// TIA Portal V21 export
FUNCTION_BLOCK "FB611"   // FB611, LAD
TITLE = FB611
{ S7_Optimized_Access := 'FALSE' }
AUTHOR : PRECISE
FAMILY : PRECISE
// CIP AIR PURGING
// stored: AutoNumber false, SetENOAutomatically false
   VAR_INPUT
      CycleEnable : Bool;
      CycleRunning : Bool;
      SecPulse : Bool;
      AlwaysTrue : Bool;
      ActualTemperature : Real;
      ActualPressure : Real;
      ActualRepetition : Int;
      ParaIn : "AirPurgingInputs";
   END_VAR
   VAR_OUTPUT
      Started : Bool;
      UtilityValve : Bool;   // Air Utility
      VentValve : Bool;
      ParaOut : "AirPurgingOutputs";
      StepStatus : String[60];
      TempValve : Bool;
      TempValve_close : Bool;
   END_VAR
   VAR_IN_OUT
      Over : Bool;
      OverTemp : Bool;
      PressurePostiveTol : Real;
      PressureNegativeTol : Real;
      ControlStarted : Bool;
      TempPostiveTol : Real;
      TempNegativeTol : Real;
      HotAirValve : Bool;
      PopupSel : Bool;
      Popup : Bool;
      PopupAck : Bool;
      ControlStartedTemp : Bool;
      re_5 : Bool;
      TempReached : Bool;
      re_6 : Bool;
   END_VAR
   VAR
      ValveOnDelayPV : Int;
      ValveOffDelayPV : Int;
      RE1 : Bool;
      StepDelay { S7_SetPoint := 'True'} : "FB110";
      VentTimer { S7_SetPoint := 'True'} : "FB101";
   END_VAR
   VAR_TEMP   // added for the SCL form of the ladder/FBD networks
      _w1 : Bool;
      _w2 : Bool;
      _w3 : Bool;
      _w4 : Bool;
   END_VAR
BEGIN

REGION Network 1: Air Purging Started
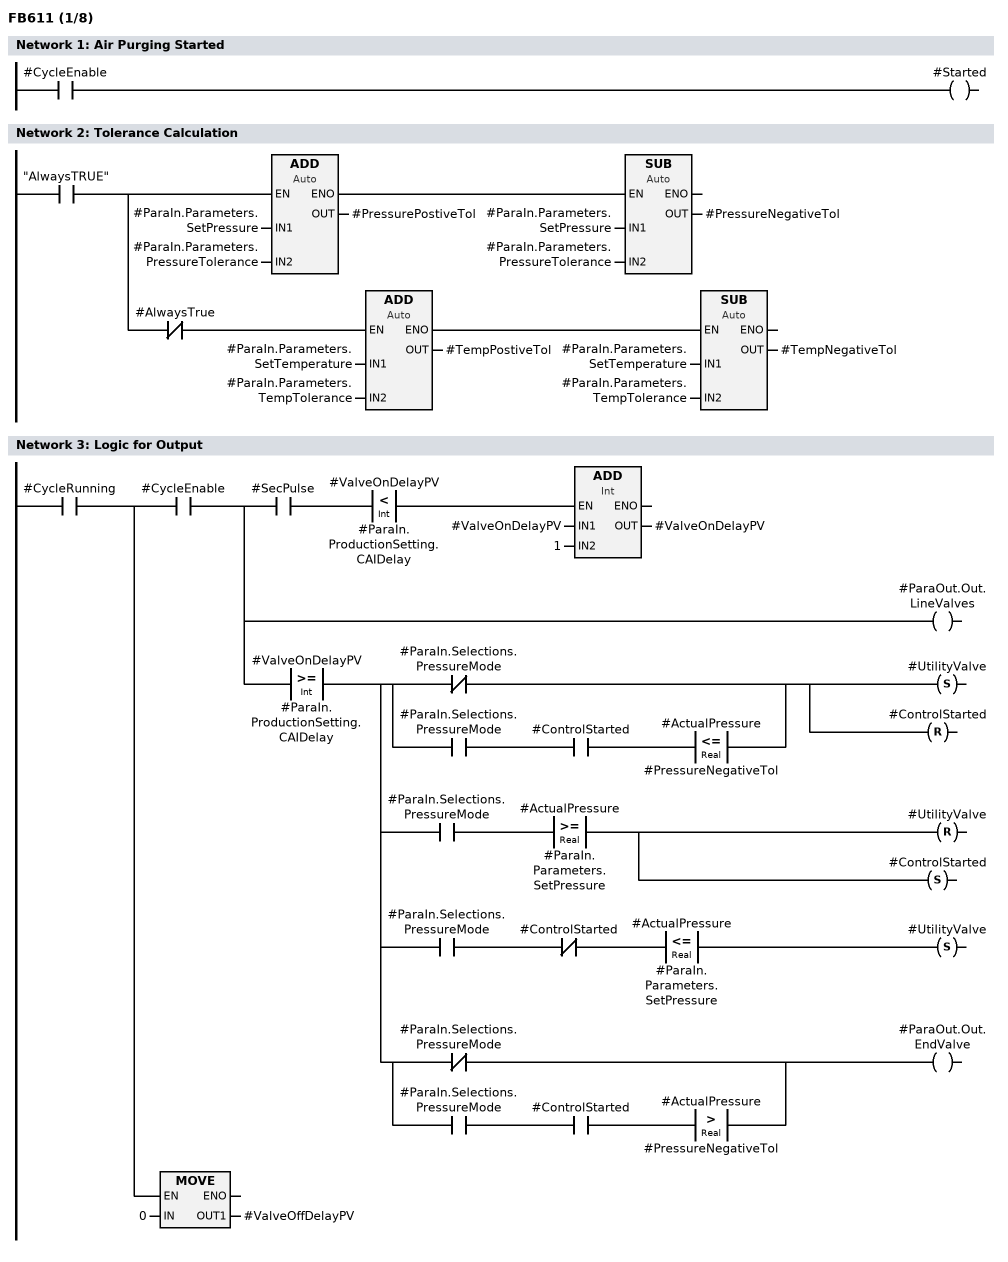
   RUNG wire#powerrail
      Contact( #CycleEnable )
      Coil( #Started )
   END_RUNG
   // the same network as SCL:
   #Started := #CycleEnable;
END_REGION

REGION Network 2: Tolerance Calculation
   RUNG wire#powerrail
      Contact( "AlwaysTRUE" )
      wire#w1
      Add(in1 := #ParaIn.Parameters.SetPressure, in2 := #ParaIn.Parameters.PressureTolerance, out => #PressurePostiveTol)
      Sub(in1 := #ParaIn.Parameters.SetPressure, in2 := #ParaIn.Parameters.PressureTolerance, out => #PressureNegativeTol)
   END_RUNG
   RUNG wire#w1
      I_Contact( #AlwaysTrue )
      Add(in1 := #ParaIn.Parameters.SetTemperature, in2 := #ParaIn.Parameters.TempTolerance, out => #TempPostiveTol)
      Sub(in1 := #ParaIn.Parameters.SetTemperature, in2 := #ParaIn.Parameters.TempTolerance, out => #TempNegativeTol)
   END_RUNG
   // the same network as SCL:
   IF "AlwaysTRUE" THEN
       #PressurePostiveTol := #ParaIn.Parameters.SetPressure + #ParaIn.Parameters.PressureTolerance;
       #PressureNegativeTol := #ParaIn.Parameters.SetPressure - #ParaIn.Parameters.PressureTolerance;
   END_IF;
   IF "AlwaysTRUE" AND NOT #AlwaysTrue THEN
       #TempPostiveTol := #ParaIn.Parameters.SetTemperature + #ParaIn.Parameters.TempTolerance;
       #TempNegativeTol := #ParaIn.Parameters.SetTemperature - #ParaIn.Parameters.TempTolerance;
   END_IF;
END_REGION

REGION Network 3: Logic for Output
   RUNG wire#powerrail
      Contact( #CycleRunning )
      wire#w1
      Contact( #CycleEnable )
      wire#w2
      Contact( #SecPulse )
      { S7_Templates := "SrcType := Int" } LT_Contact(in1 := #ValveOnDelayPV, in2 := #ParaIn.ProductionSetting.CAIDelay)
      { S7_Templates := "SrcType := Int"; S7_GenerateENO := "TRUE" } Add(in1 := #ValveOnDelayPV, in2 := 1, out => #ValveOnDelayPV)
   END_RUNG
   RUNG wire#w2
      Coil( #ParaOut.Out.LineValves )
   END_RUNG
   RUNG wire#w2
      { S7_Templates := "SrcType := Int" } GE_Contact(in1 := #ValveOnDelayPV, in2 := #ParaIn.ProductionSetting.CAIDelay)
      wire#w3
      I_Contact( #ParaIn.Selections.PressureMode )
      wire#w4
      S_Coil( #UtilityValve )
   END_RUNG
   RUNG wire#w3
      Contact( #ParaIn.Selections.PressureMode )
      Contact( #ControlStarted )
      { S7_Templates := "SrcType := Real" } LE_Contact(in1 := #ActualPressure, in2 := #PressureNegativeTol)
   END_RUNG wire#w4
   RUNG wire#w4
      R_Coil( #ControlStarted )
   END_RUNG
   RUNG wire#w3
      Contact( #ParaIn.Selections.PressureMode )
      { S7_Templates := "SrcType := Real" } GE_Contact(in1 := #ActualPressure, in2 := #ParaIn.Parameters.SetPressure)
      wire#w5
      R_Coil( #UtilityValve )
   END_RUNG
   RUNG wire#w5
      S_Coil( #ControlStarted )
   END_RUNG
   RUNG wire#w3
      Contact( #ParaIn.Selections.PressureMode )
      I_Contact( #ControlStarted )
      { S7_Templates := "SrcType := Real" } LE_Contact(in1 := #ActualPressure, in2 := #ParaIn.Parameters.SetPressure)
      S_Coil( #UtilityValve )
   END_RUNG
   RUNG wire#w3
      I_Contact( #ParaIn.Selections.PressureMode )
      wire#w6
      Coil( #ParaOut.Out.EndValve )
   END_RUNG
   RUNG wire#w3
      Contact( #ParaIn.Selections.PressureMode )
      Contact( #ControlStarted )
      { S7_Templates := "SrcType := Real" } GT_Contact(in1 := #ActualPressure, in2 := #PressureNegativeTol)
   END_RUNG wire#w6
   RUNG wire#w1
      { S7_GenerateENO := "TRUE" } Move(in := 0, out1 => #ValveOffDelayPV)
   END_RUNG
   // the same network as SCL:
   #_w1 := #CycleRunning AND #CycleEnable;
   IF #_w1 AND #SecPulse AND (#ValveOnDelayPV < #ParaIn.ProductionSetting.CAIDelay) THEN
       #ValveOnDelayPV := #ValveOnDelayPV + 1;
   END_IF;
   #ParaOut.Out.LineValves := #_w1;
   #_w2 := #_w1 AND (#ValveOnDelayPV >= #ParaIn.ProductionSetting.CAIDelay);
   IF #_w2 AND (NOT #ParaIn.Selections.PressureMode OR (#ParaIn.Selections.PressureMode AND #ControlStarted AND (#ActualPressure <= #PressureNegativeTol))) THEN
       #UtilityValve := TRUE;
       #ControlStarted := FALSE;
   END_IF;
   IF #_w2 AND #ParaIn.Selections.PressureMode AND (#ActualPressure >= #ParaIn.Parameters.SetPressure) THEN
       #UtilityValve := FALSE;
       #ControlStarted := TRUE;
   END_IF;
   IF #_w2 AND #ParaIn.Selections.PressureMode AND NOT #ControlStarted AND (#ActualPressure <= #ParaIn.Parameters.SetPressure) THEN
       #UtilityValve := TRUE;
   END_IF;
   #ParaOut.Out.EndValve := #_w2 AND (NOT #ParaIn.Selections.PressureMode OR (#ParaIn.Selections.PressureMode AND #ControlStarted AND (#ActualPressure > #PressureNegativeTol)));
   IF #CycleRunning THEN #ValveOffDelayPV := 0; END_IF;
END_REGION

REGION Network 4: Logic for Output Air Purging Sel
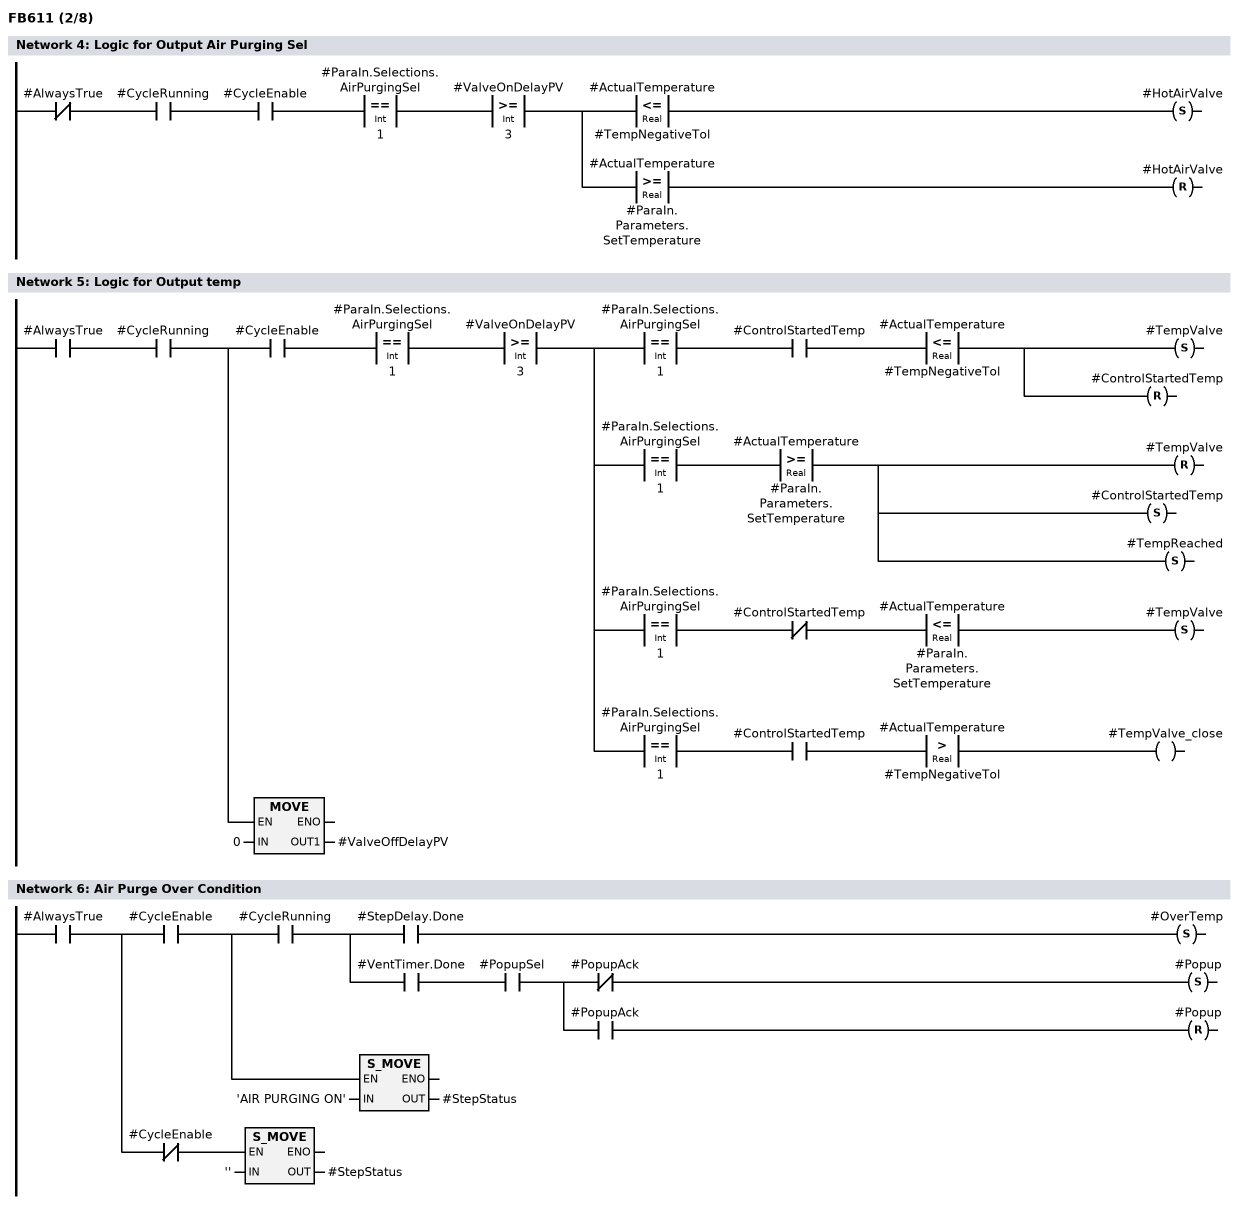
   RUNG wire#powerrail
      I_Contact( #AlwaysTrue )
      Contact( #CycleRunning )
      Contact( #CycleEnable )
      { S7_Templates := "SrcType := Int" } EQ_Contact(in1 := #ParaIn.Selections.AirPurgingSel, in2 := 1)
      { S7_Templates := "SrcType := Int" } GE_Contact(in1 := #ValveOnDelayPV, in2 := 3)
      wire#w1
      { S7_Templates := "SrcType := Real" } LE_Contact(in1 := #ActualTemperature, in2 := #TempNegativeTol)
      S_Coil( #HotAirValve )
   END_RUNG
   RUNG wire#w1
      { S7_Templates := "SrcType := Real" } GE_Contact(in1 := #ActualTemperature, in2 := #ParaIn.Parameters.SetTemperature)
      R_Coil( #HotAirValve )
   END_RUNG
   // the same network as SCL:
   #_w1 := NOT #AlwaysTrue AND #CycleRunning AND #CycleEnable AND (#ParaIn.Selections.AirPurgingSel = 1) AND (#ValveOnDelayPV >= 3);
   IF #_w1 AND (#ActualTemperature <= #TempNegativeTol) THEN #HotAirValve := TRUE; END_IF;
   IF #_w1 AND (#ActualTemperature >= #ParaIn.Parameters.SetTemperature) THEN #HotAirValve := FALSE; END_IF;
END_REGION

REGION Network 5: Logic for Output temp
   RUNG wire#powerrail
      Contact( #AlwaysTrue )
      Contact( #CycleRunning )
      wire#w1
      Contact( #CycleEnable )
      { S7_Templates := "SrcType := Int" } EQ_Contact(in1 := #ParaIn.Selections.AirPurgingSel, in2 := 1)
      { S7_Templates := "SrcType := Int" } GE_Contact(in1 := #ValveOnDelayPV, in2 := 3)
      wire#w2
      { S7_Templates := "SrcType := Int" } EQ_Contact(in1 := #ParaIn.Selections.AirPurgingSel, in2 := 1)
      Contact( #ControlStartedTemp )
      { S7_Templates := "SrcType := Real" } LE_Contact(in1 := #ActualTemperature, in2 := #TempNegativeTol)
      wire#w3
      S_Coil( #TempValve )
   END_RUNG
   RUNG wire#w3
      R_Coil( #ControlStartedTemp )
   END_RUNG
   RUNG wire#w2
      { S7_Templates := "SrcType := Int" } EQ_Contact(in1 := #ParaIn.Selections.AirPurgingSel, in2 := 1)
      { S7_Templates := "SrcType := Real" } GE_Contact(in1 := #ActualTemperature, in2 := #ParaIn.Parameters.SetTemperature)
      wire#w4
      R_Coil( #TempValve )
   END_RUNG
   RUNG wire#w4
      S_Coil( #ControlStartedTemp )
   END_RUNG
   RUNG wire#w4
      S_Coil( #TempReached )
   END_RUNG
   RUNG wire#w2
      { S7_Templates := "SrcType := Int" } EQ_Contact(in1 := #ParaIn.Selections.AirPurgingSel, in2 := 1)
      I_Contact( #ControlStartedTemp )
      { S7_Templates := "SrcType := Real" } LE_Contact(in1 := #ActualTemperature, in2 := #ParaIn.Parameters.SetTemperature)
      S_Coil( #TempValve )
   END_RUNG
   RUNG wire#w2
      { S7_Templates := "SrcType := Int" } EQ_Contact(in1 := #ParaIn.Selections.AirPurgingSel, in2 := 1)
      Contact( #ControlStartedTemp )
      { S7_Templates := "SrcType := Real" } GT_Contact(in1 := #ActualTemperature, in2 := #TempNegativeTol)
      Coil( #TempValve_close )
   END_RUNG
   RUNG wire#w1
      { S7_GenerateENO := "TRUE" } Move(in := 0, out1 => #ValveOffDelayPV)
   END_RUNG
   // the same network as SCL:
   #_w1 := #AlwaysTrue AND #CycleRunning;
   #_w2 := #_w1 AND #CycleEnable AND (#ParaIn.Selections.AirPurgingSel = 1) AND (#ValveOnDelayPV >= 3);
   IF #_w2 AND (#ParaIn.Selections.AirPurgingSel = 1) AND #ControlStartedTemp AND (#ActualTemperature <= #TempNegativeTol) THEN
       #TempValve := TRUE;
       #ControlStartedTemp := FALSE;
   END_IF;
   IF #_w2 AND (#ParaIn.Selections.AirPurgingSel = 1) AND (#ActualTemperature >= #ParaIn.Parameters.SetTemperature) THEN
       #TempValve := FALSE;
       #ControlStartedTemp := TRUE;
       #TempReached := TRUE;
   END_IF;
   IF #_w2 AND (#ParaIn.Selections.AirPurgingSel = 1) AND NOT #ControlStartedTemp AND (#ActualTemperature <= #ParaIn.Parameters.SetTemperature) THEN
       #TempValve := TRUE;
   END_IF;
   #TempValve_close := #_w2 AND (#ParaIn.Selections.AirPurgingSel = 1) AND #ControlStartedTemp AND (#ActualTemperature > #TempNegativeTol);
   IF #_w1 THEN #ValveOffDelayPV := 0; END_IF;
END_REGION

REGION Network 6: Air Purge Over Condition
   RUNG wire#powerrail
      Contact( #AlwaysTrue )
      wire#w1
      Contact( #CycleEnable )
      wire#w2
      Contact( #CycleRunning )
      wire#w3
      Contact( #StepDelay.Done )
      S_Coil( #OverTemp )
   END_RUNG
   RUNG wire#w3
      Contact( #VentTimer.Done )
      Contact( #PopupSel )
      wire#w4
      I_Contact( #PopupAck )
      S_Coil( #Popup )
   END_RUNG
   RUNG wire#w4
      Contact( #PopupAck )
      R_Coil( #Popup )
   END_RUNG
   RUNG wire#w2
      S_Move(in := 'AIR PURGING ON', out => #StepStatus)
   END_RUNG
   RUNG wire#w1
      I_Contact( #CycleEnable )
      S_Move(in := '', out => #StepStatus)
   END_RUNG
   // the same network as SCL:
   #_w1 := #AlwaysTrue AND #CycleEnable;
   #_w2 := #_w1 AND #CycleRunning;
   IF #_w2 AND #StepDelay.Done THEN #OverTemp := TRUE; END_IF;
   #_w3 := #_w2 AND #VentTimer.Done AND #PopupSel;
   IF #_w3 AND NOT #PopupAck THEN #Popup := TRUE; END_IF;
   IF #_w3 AND #PopupAck THEN #Popup := FALSE; END_IF;
   IF #_w1 THEN #StepStatus := 'AIR PURGING ON'; END_IF;
   IF #AlwaysTrue AND NOT #CycleEnable THEN #StepStatus := ''; END_IF;
END_REGION

REGION Network 7: Air Purge Over
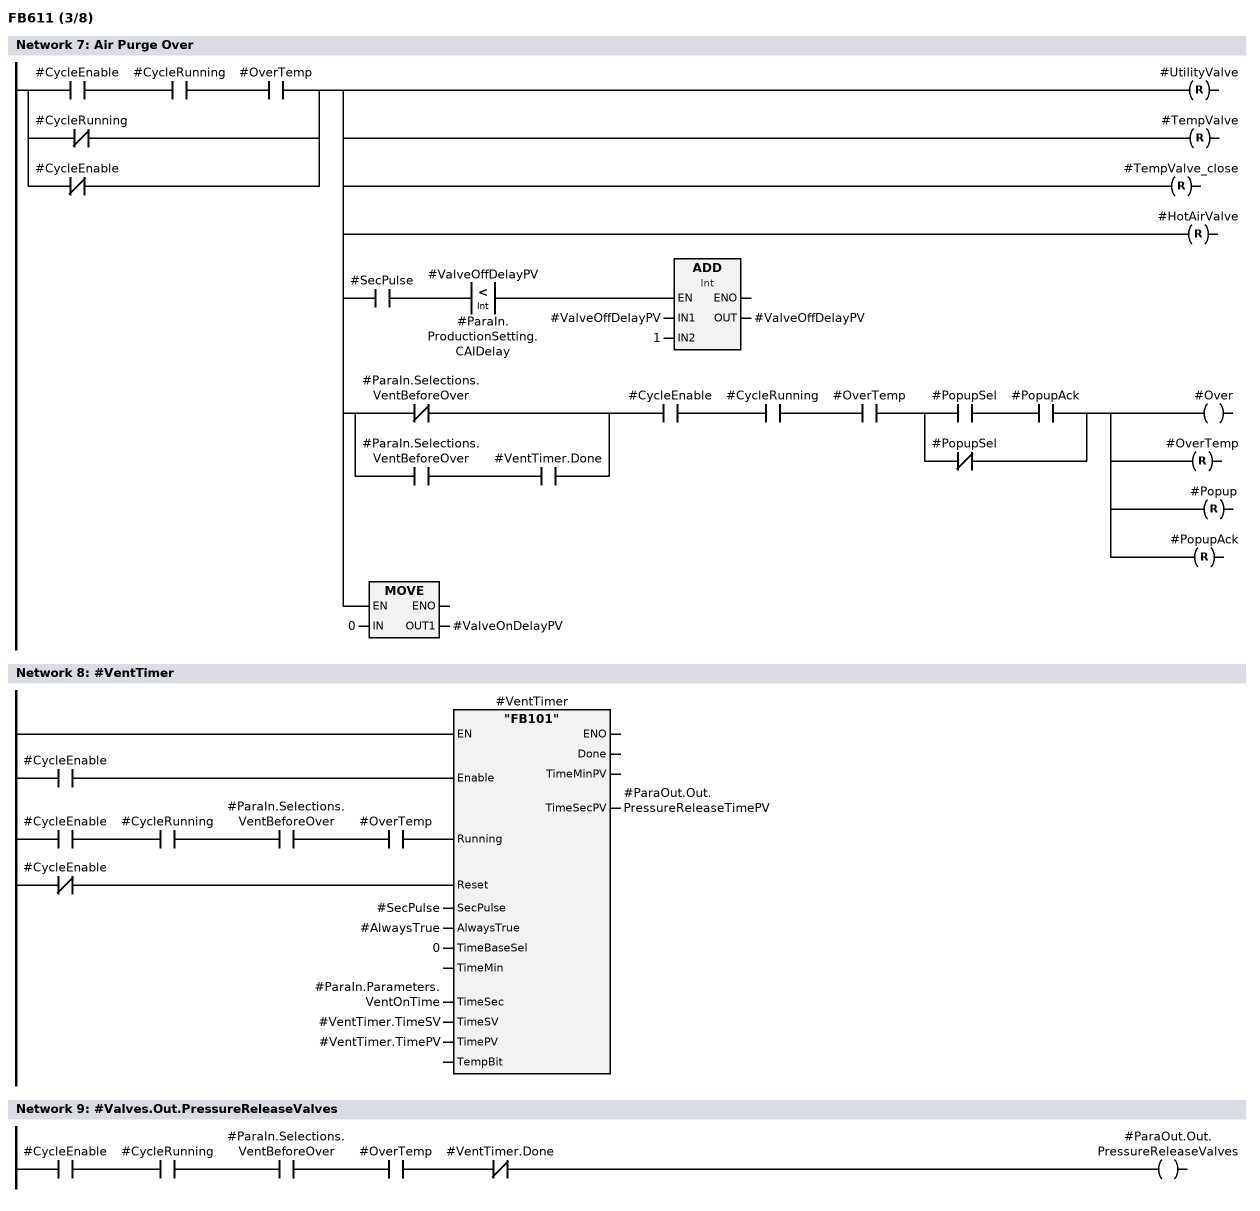
   RUNG wire#powerrail
      Contact( #CycleEnable )
      Contact( #CycleRunning )
      Contact( #OverTemp )
      wire#w1
      R_Coil( #UtilityValve )
   END_RUNG
   RUNG wire#powerrail
      I_Contact( #CycleRunning )
   END_RUNG wire#w1
   RUNG wire#powerrail
      I_Contact( #CycleEnable )
   END_RUNG wire#w1
   RUNG wire#w1
      R_Coil( #TempValve )
   END_RUNG
   RUNG wire#w1
      R_Coil( #TempValve_close )
   END_RUNG
   RUNG wire#w1
      R_Coil( #HotAirValve )
   END_RUNG
   RUNG wire#w1
      Contact( #SecPulse )
      { S7_Templates := "SrcType := Int" } LT_Contact(in1 := #ValveOffDelayPV, in2 := #ParaIn.ProductionSetting.CAIDelay)
      { S7_Templates := "SrcType := Int"; S7_GenerateENO := "TRUE" } Add(in1 := #ValveOffDelayPV, in2 := 1, out => #ValveOffDelayPV)
   END_RUNG
   RUNG wire#w1
      I_Contact( #ParaIn.Selections.VentBeforeOver )
      wire#w2
      Contact( #CycleEnable )
      Contact( #CycleRunning )
      Contact( #OverTemp )
      wire#w3
      Contact( #PopupSel )
      Contact( #PopupAck )
      wire#w4
      Coil( #Over )
   END_RUNG
   RUNG wire#w1
      Contact( #ParaIn.Selections.VentBeforeOver )
      Contact( #VentTimer.Done )
   END_RUNG wire#w2
   RUNG wire#w3
      I_Contact( #PopupSel )
   END_RUNG wire#w4
   RUNG wire#w4
      R_Coil( #OverTemp )
   END_RUNG
   RUNG wire#w4
      R_Coil( #Popup )
   END_RUNG
   RUNG wire#w4
      R_Coil( #PopupAck )
   END_RUNG
   RUNG wire#w1
      { S7_GenerateENO := "TRUE" } Move(in := 0, out1 => #ValveOnDelayPV)
   END_RUNG
   // the same network as SCL:
   #_w1 := (#CycleEnable AND #CycleRunning AND #OverTemp) OR NOT #CycleRunning OR NOT #CycleEnable;
   IF #_w1 THEN
       #UtilityValve := FALSE;
       #TempValve := FALSE;
       #TempValve_close := FALSE;
       #HotAirValve := FALSE;
   END_IF;
   IF #_w1 AND #SecPulse AND (#ValveOffDelayPV < #ParaIn.ProductionSetting.CAIDelay) THEN
       #ValveOffDelayPV := #ValveOffDelayPV + 1;
   END_IF;
   #Over := #_w1 AND (NOT #ParaIn.Selections.VentBeforeOver OR (#ParaIn.Selections.VentBeforeOver AND #VentTimer.Done)) AND #CycleEnable AND #CycleRunning AND #OverTemp AND ((#PopupSel AND #PopupAck) OR NOT #PopupSel);
   IF #Over THEN
       #OverTemp := FALSE;
       #Popup := FALSE;
       #PopupAck := FALSE;
   END_IF;
   IF #_w1 THEN #ValveOnDelayPV := 0; END_IF;
END_REGION

REGION Network 8: #VentTimer
   RUNG wire#powerrail
      #VentTimer(Enable := wire#w1, Running := wire#w2, Reset := wire#w3, SecPulse := #SecPulse, AlwaysTrue := #AlwaysTrue, TimeBaseSel := 0, TimeMin :=, TimeSec := #ParaIn.Parameters.VentOnTime, TimeSV := #VentTimer.TimeSV, TimePV := #VentTimer.TimePV, TempBit :=, Done =>, TimeMinPV =>, TimeSecPV => #ParaOut.Out.PressureReleaseTimePV)
   END_RUNG
   RUNG wire#powerrail
      Contact( #CycleEnable )
   END_RUNG wire#w1
   RUNG wire#powerrail
      Contact( #CycleEnable )
      Contact( #CycleRunning )
      Contact( #ParaIn.Selections.VentBeforeOver )
      Contact( #OverTemp )
   END_RUNG wire#w2
   RUNG wire#powerrail
      I_Contact( #CycleEnable )
   END_RUNG wire#w3
   // the same network as SCL:
   #VentTimer(Enable := #CycleEnable,   // "FB101"
              Running := #CycleEnable AND #CycleRunning AND #ParaIn.Selections.VentBeforeOver AND #OverTemp,
              Reset := NOT #CycleEnable,
              SecPulse := #SecPulse,
              AlwaysTrue := #AlwaysTrue,
              TimeBaseSel := 0,
              TimeSec := #ParaIn.Parameters.VentOnTime,
              TimeSV := #VentTimer.TimeSV,
              TimePV := #VentTimer.TimePV,
              TimeSecPV => #ParaOut.Out.PressureReleaseTimePV);
END_REGION

REGION Network 9: #Valves.Out.PressureReleaseValves
   RUNG wire#powerrail
      Contact( #CycleEnable )
      Contact( #CycleRunning )
      Contact( #ParaIn.Selections.VentBeforeOver )
      Contact( #OverTemp )
      I_Contact( #VentTimer.Done )
      Coil( #ParaOut.Out.PressureReleaseValves )
   END_RUNG
   // the same network as SCL:
   #ParaOut.Out.PressureReleaseValves := #CycleEnable AND #CycleRunning AND #ParaIn.Selections.VentBeforeOver AND #OverTemp AND NOT #VentTimer.Done;
END_REGION

REGION Network 10: StepDelay.StepTimeSV
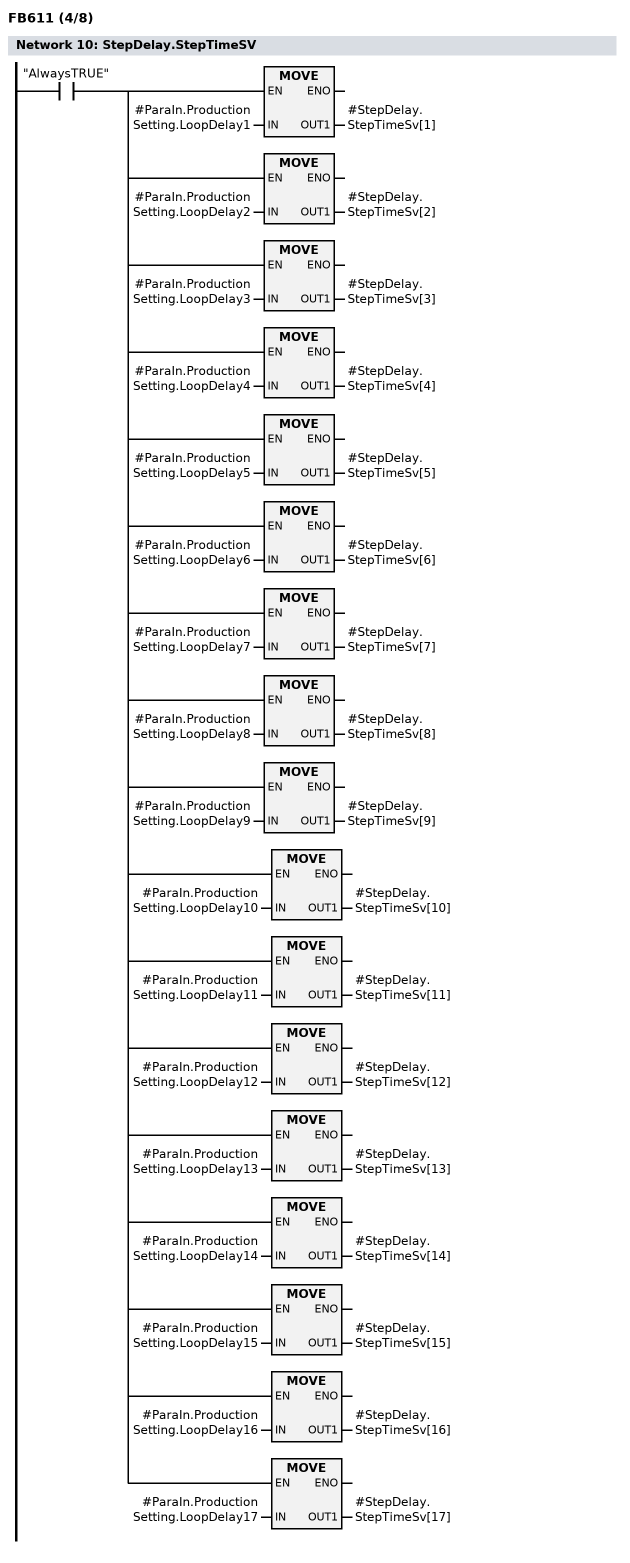
   RUNG wire#powerrail
      Contact( "AlwaysTRUE" )
      wire#w1
      Move(in := #ParaIn.ProductionSetting.LoopDelay1, out1 => #StepDelay.StepTimeSv[1])
   END_RUNG
   RUNG wire#w1
      Move(in := #ParaIn.ProductionSetting.LoopDelay2, out1 => #StepDelay.StepTimeSv[2])
   END_RUNG
   RUNG wire#w1
      Move(in := #ParaIn.ProductionSetting.LoopDelay3, out1 => #StepDelay.StepTimeSv[3])
   END_RUNG
   RUNG wire#w1
      Move(in := #ParaIn.ProductionSetting.LoopDelay4, out1 => #StepDelay.StepTimeSv[4])
   END_RUNG
   RUNG wire#w1
      Move(in := #ParaIn.ProductionSetting.LoopDelay5, out1 => #StepDelay.StepTimeSv[5])
   END_RUNG
   RUNG wire#w1
      Move(in := #ParaIn.ProductionSetting.LoopDelay6, out1 => #StepDelay.StepTimeSv[6])
   END_RUNG
   RUNG wire#w1
      Move(in := #ParaIn.ProductionSetting.LoopDelay7, out1 => #StepDelay.StepTimeSv[7])
   END_RUNG
   RUNG wire#w1
      Move(in := #ParaIn.ProductionSetting.LoopDelay8, out1 => #StepDelay.StepTimeSv[8])
   END_RUNG
   RUNG wire#w1
      Move(in := #ParaIn.ProductionSetting.LoopDelay9, out1 => #StepDelay.StepTimeSv[9])
   END_RUNG
   RUNG wire#w1
      Move(in := #ParaIn.ProductionSetting.LoopDelay10, out1 => #StepDelay.StepTimeSv[10])
   END_RUNG
   RUNG wire#w1
      Move(in := #ParaIn.ProductionSetting.LoopDelay11, out1 => #StepDelay.StepTimeSv[11])
   END_RUNG
   RUNG wire#w1
      Move(in := #ParaIn.ProductionSetting.LoopDelay12, out1 => #StepDelay.StepTimeSv[12])
   END_RUNG
   RUNG wire#w1
      Move(in := #ParaIn.ProductionSetting.LoopDelay13, out1 => #StepDelay.StepTimeSv[13])
   END_RUNG
   RUNG wire#w1
      Move(in := #ParaIn.ProductionSetting.LoopDelay14, out1 => #StepDelay.StepTimeSv[14])
   END_RUNG
   RUNG wire#w1
      Move(in := #ParaIn.ProductionSetting.LoopDelay15, out1 => #StepDelay.StepTimeSv[15])
   END_RUNG
   RUNG wire#w1
      Move(in := #ParaIn.ProductionSetting.LoopDelay16, out1 => #StepDelay.StepTimeSv[16])
   END_RUNG
   RUNG wire#w1
      Move(in := #ParaIn.ProductionSetting.LoopDelay17, out1 => #StepDelay.StepTimeSv[17])
   END_RUNG
   // the same network as SCL:
   IF "AlwaysTRUE" THEN
       #StepDelay.StepTimeSv[1] := #ParaIn.ProductionSetting.LoopDelay1;
       #StepDelay.StepTimeSv[2] := #ParaIn.ProductionSetting.LoopDelay2;
       #StepDelay.StepTimeSv[3] := #ParaIn.ProductionSetting.LoopDelay3;
       #StepDelay.StepTimeSv[4] := #ParaIn.ProductionSetting.LoopDelay4;
       #StepDelay.StepTimeSv[5] := #ParaIn.ProductionSetting.LoopDelay5;
       #StepDelay.StepTimeSv[6] := #ParaIn.ProductionSetting.LoopDelay6;
       #StepDelay.StepTimeSv[7] := #ParaIn.ProductionSetting.LoopDelay7;
       #StepDelay.StepTimeSv[8] := #ParaIn.ProductionSetting.LoopDelay8;
       #StepDelay.StepTimeSv[9] := #ParaIn.ProductionSetting.LoopDelay9;
       #StepDelay.StepTimeSv[10] := #ParaIn.ProductionSetting.LoopDelay10;
       #StepDelay.StepTimeSv[11] := #ParaIn.ProductionSetting.LoopDelay11;
       #StepDelay.StepTimeSv[12] := #ParaIn.ProductionSetting.LoopDelay12;
       #StepDelay.StepTimeSv[13] := #ParaIn.ProductionSetting.LoopDelay13;
       #StepDelay.StepTimeSv[14] := #ParaIn.ProductionSetting.LoopDelay14;
       #StepDelay.StepTimeSv[15] := #ParaIn.ProductionSetting.LoopDelay15;
       #StepDelay.StepTimeSv[16] := #ParaIn.ProductionSetting.LoopDelay16;
       #StepDelay.StepTimeSv[17] := #ParaIn.ProductionSetting.LoopDelay17;
   END_IF;
END_REGION

REGION Network 11: sv and pv for run screen
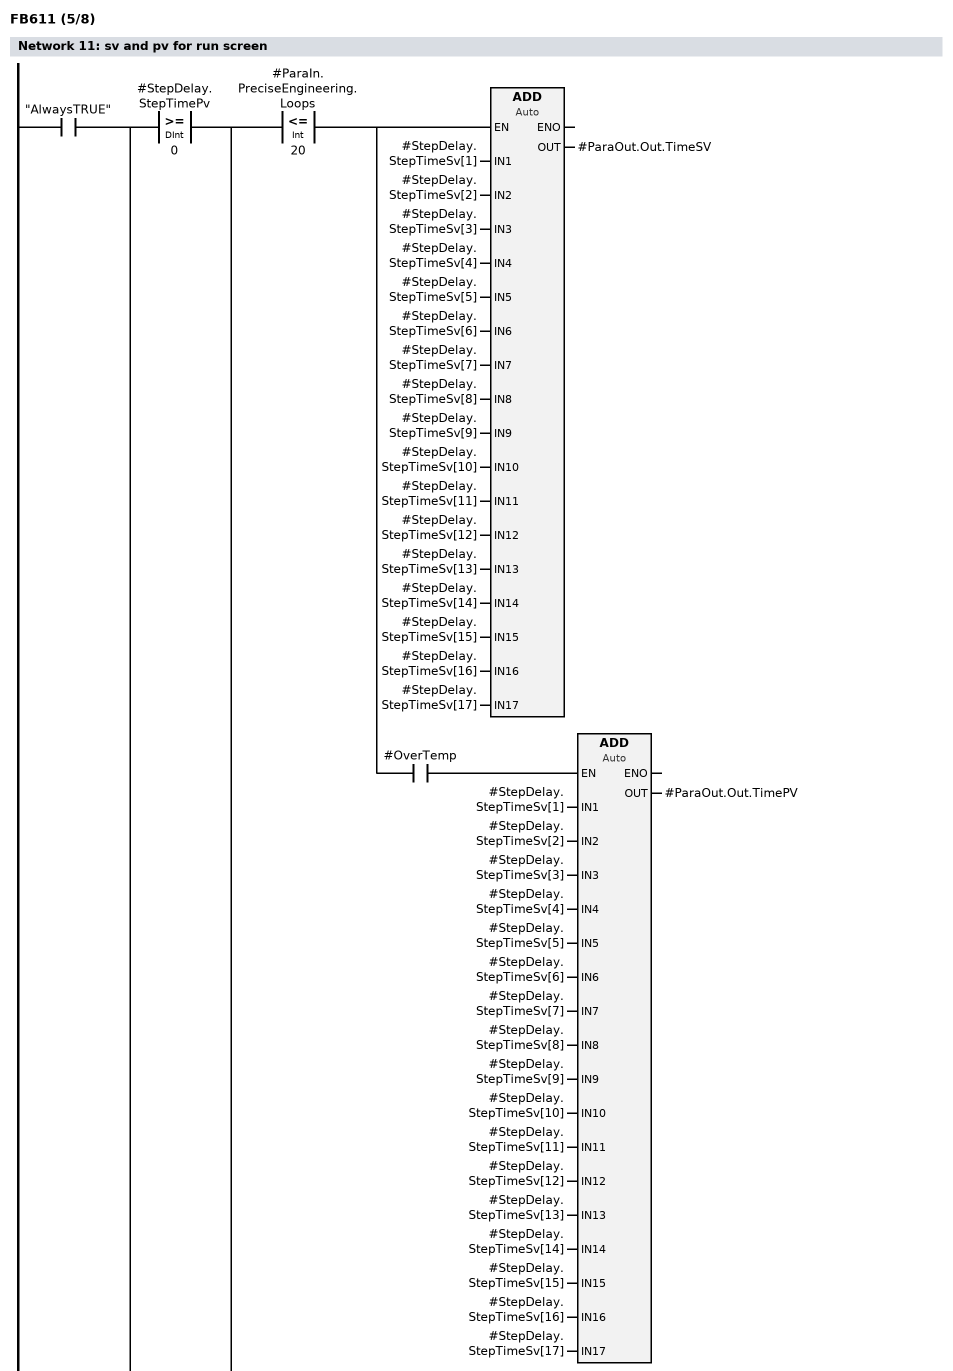
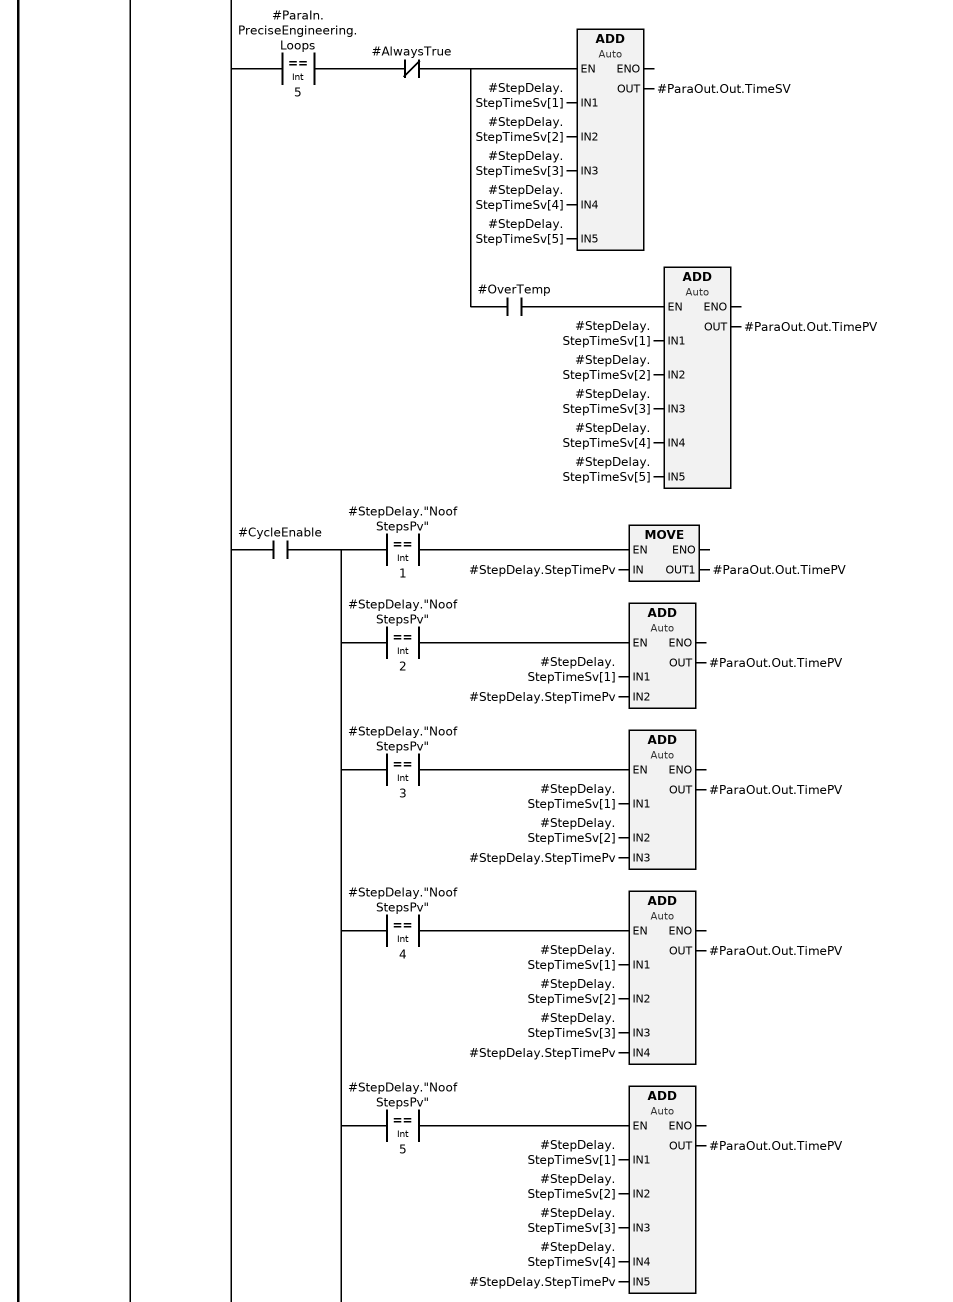
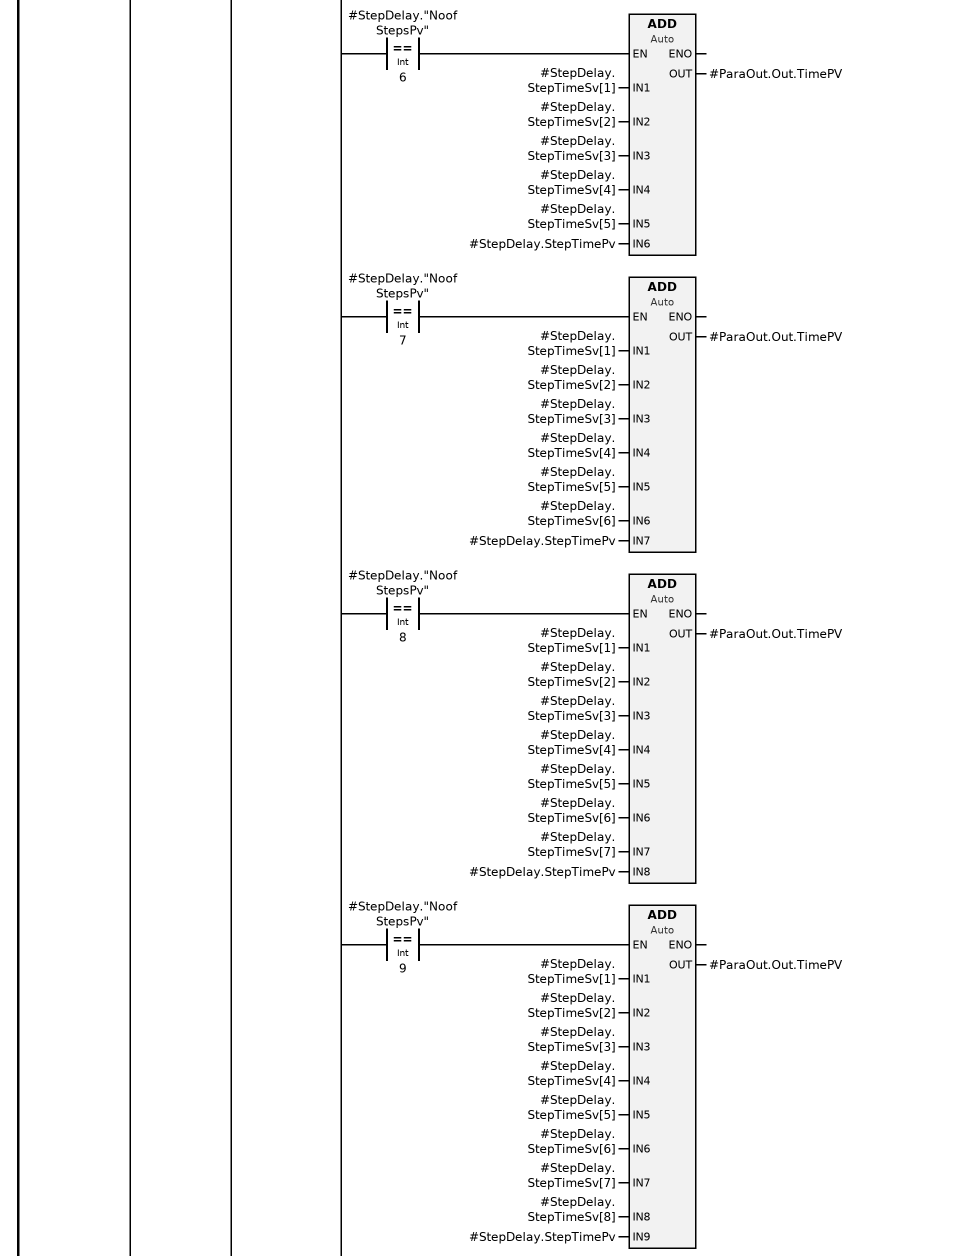
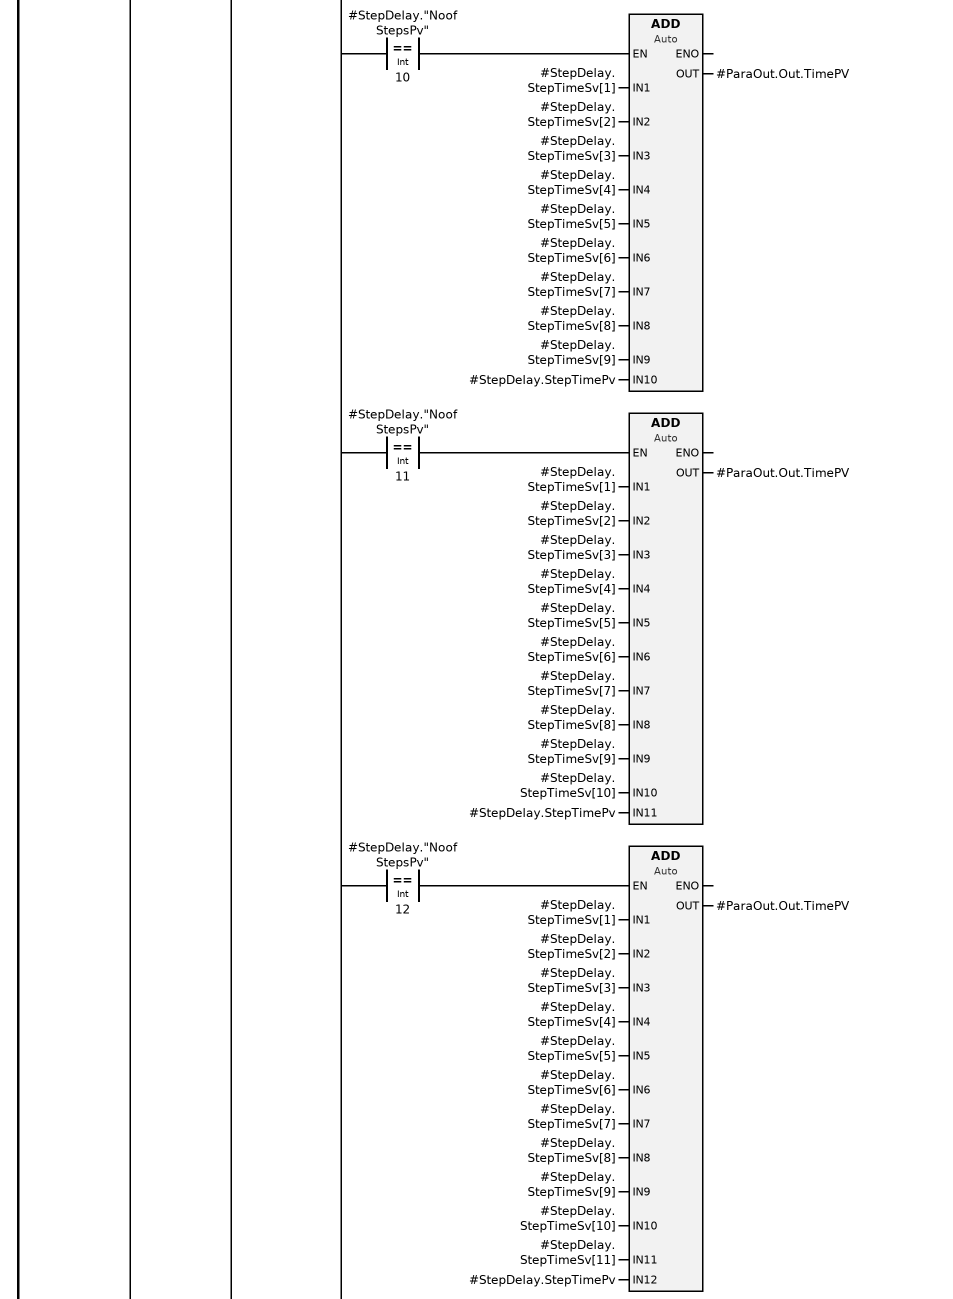
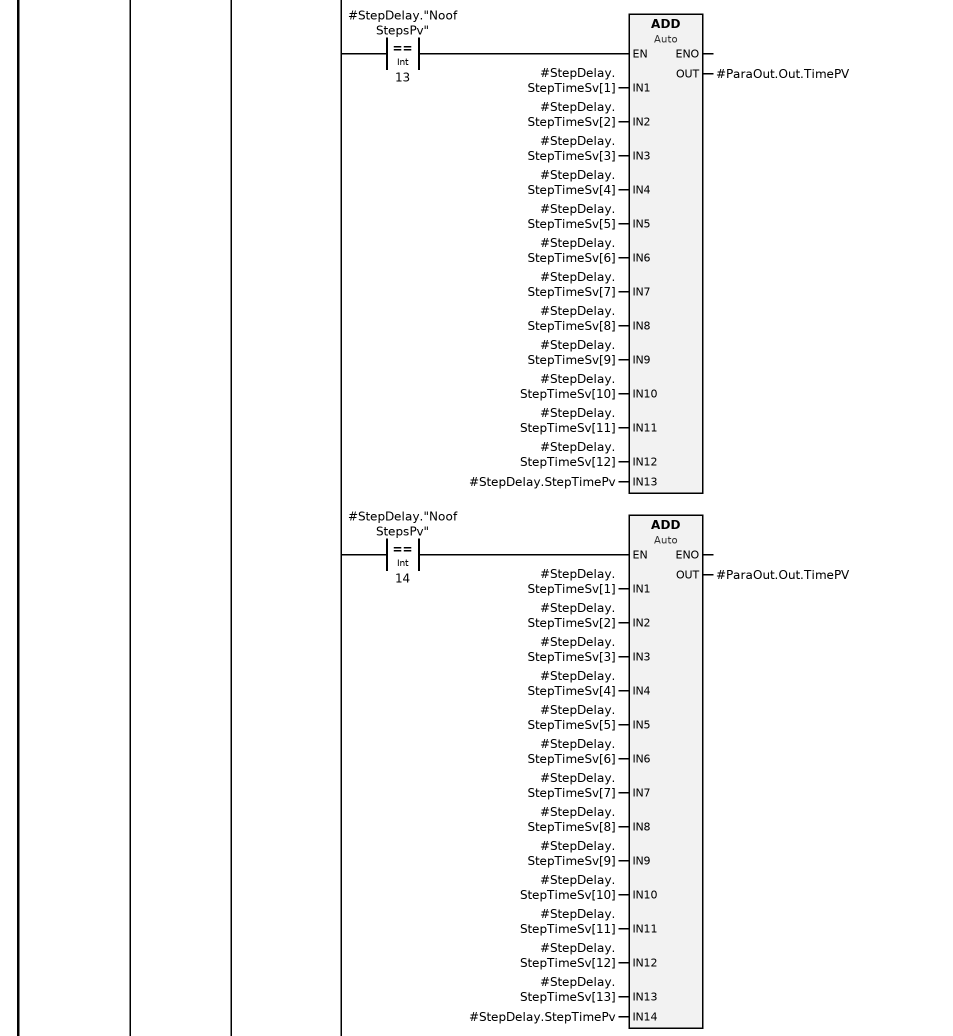
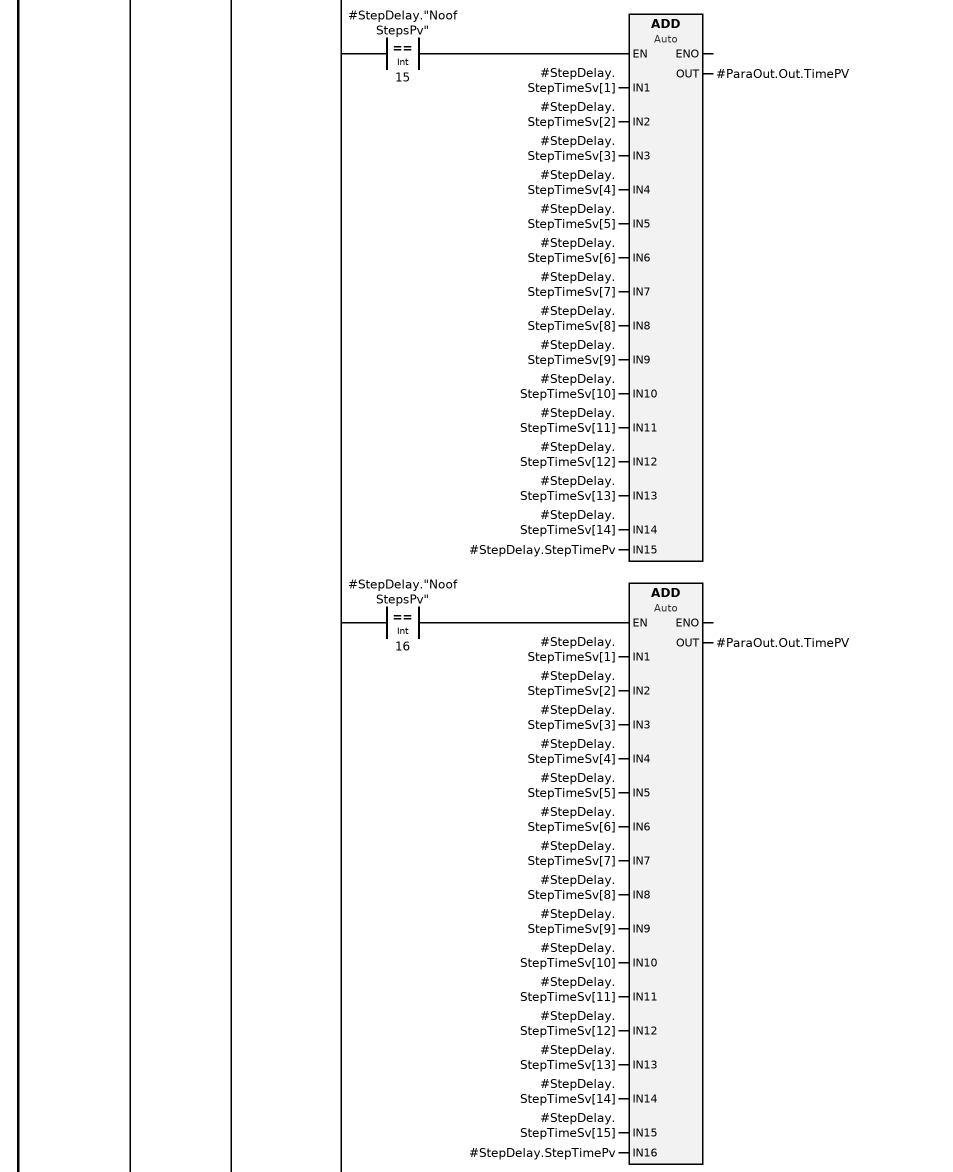
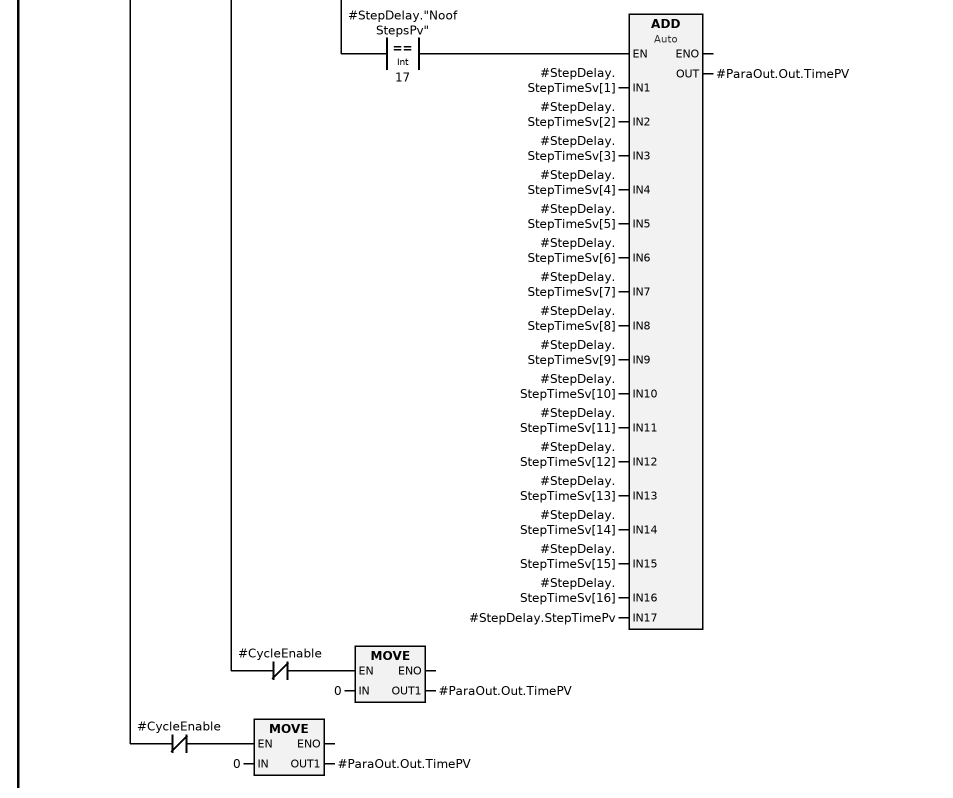
   RUNG wire#powerrail
      Contact( "AlwaysTRUE" )
      wire#w1
      { S7_Templates := "SrcType := DInt" } GE_Contact(in1 := #StepDelay.StepTimePv, in2 := 0)
      wire#w2
      { S7_Templates := "SrcType := Int" } LE_Contact(in1 := #ParaIn.PreciseEngineering.Loops, in2 := 20)
      wire#w3
      Add(in1 := #StepDelay.StepTimeSv[1], in2 := #StepDelay.StepTimeSv[2], in3 := #StepDelay.StepTimeSv[3], in4 := #StepDelay.StepTimeSv[4], in5 := #StepDelay.StepTimeSv[5], in6 := #StepDelay.StepTimeSv[6], in7 := #StepDelay.StepTimeSv[7], in8 := #StepDelay.StepTimeSv[8], in9 := #StepDelay.StepTimeSv[9], in10 := #StepDelay.StepTimeSv[10], in11 := #StepDelay.StepTimeSv[11], in12 := #StepDelay.StepTimeSv[12], in13 := #StepDelay.StepTimeSv[13], in14 := #StepDelay.StepTimeSv[14], in15 := #StepDelay.StepTimeSv[15], in16 := #StepDelay.StepTimeSv[16], in17 := #StepDelay.StepTimeSv[17], out => #ParaOut.Out.TimeSV)
   END_RUNG
   RUNG wire#w3
      Contact( #OverTemp )
      Add(in1 := #StepDelay.StepTimeSv[1], in2 := #StepDelay.StepTimeSv[2], in3 := #StepDelay.StepTimeSv[3], in4 := #StepDelay.StepTimeSv[4], in5 := #StepDelay.StepTimeSv[5], in6 := #StepDelay.StepTimeSv[6], in7 := #StepDelay.StepTimeSv[7], in8 := #StepDelay.StepTimeSv[8], in9 := #StepDelay.StepTimeSv[9], in10 := #StepDelay.StepTimeSv[10], in11 := #StepDelay.StepTimeSv[11], in12 := #StepDelay.StepTimeSv[12], in13 := #StepDelay.StepTimeSv[13], in14 := #StepDelay.StepTimeSv[14], in15 := #StepDelay.StepTimeSv[15], in16 := #StepDelay.StepTimeSv[16], in17 := #StepDelay.StepTimeSv[17], out => #ParaOut.Out.TimePV)
   END_RUNG
   RUNG wire#w2
      { S7_Templates := "SrcType := Int" } EQ_Contact(in1 := #ParaIn.PreciseEngineering.Loops, in2 := 5)
      I_Contact( #AlwaysTrue )
      wire#w4
      Add(in1 := #StepDelay.StepTimeSv[1], in2 := #StepDelay.StepTimeSv[2], in3 := #StepDelay.StepTimeSv[3], in4 := #StepDelay.StepTimeSv[4], in5 := #StepDelay.StepTimeSv[5], out => #ParaOut.Out.TimeSV)
   END_RUNG
   RUNG wire#w4
      Contact( #OverTemp )
      Add(in1 := #StepDelay.StepTimeSv[1], in2 := #StepDelay.StepTimeSv[2], in3 := #StepDelay.StepTimeSv[3], in4 := #StepDelay.StepTimeSv[4], in5 := #StepDelay.StepTimeSv[5], out => #ParaOut.Out.TimePV)
   END_RUNG
   RUNG wire#w2
      Contact( #CycleEnable )
      wire#w5
      { S7_Templates := "SrcType := Int" } EQ_Contact(in1 := #StepDelay."Noof StepsPv", in2 := 1)
      Move(in := #StepDelay.StepTimePv, out1 => #ParaOut.Out.TimePV)
   END_RUNG
   RUNG wire#w5
      { S7_Templates := "SrcType := Int" } EQ_Contact(in1 := #StepDelay."Noof StepsPv", in2 := 2)
      Add(in1 := #StepDelay.StepTimeSv[1], in2 := #StepDelay.StepTimePv, out => #ParaOut.Out.TimePV)
   END_RUNG
   RUNG wire#w5
      { S7_Templates := "SrcType := Int" } EQ_Contact(in1 := #StepDelay."Noof StepsPv", in2 := 3)
      Add(in1 := #StepDelay.StepTimeSv[1], in2 := #StepDelay.StepTimeSv[2], in3 := #StepDelay.StepTimePv, out => #ParaOut.Out.TimePV)
   END_RUNG
   RUNG wire#w5
      { S7_Templates := "SrcType := Int" } EQ_Contact(in1 := #StepDelay."Noof StepsPv", in2 := 4)
      Add(in1 := #StepDelay.StepTimeSv[1], in2 := #StepDelay.StepTimeSv[2], in3 := #StepDelay.StepTimeSv[3], in4 := #StepDelay.StepTimePv, out => #ParaOut.Out.TimePV)
   END_RUNG
   RUNG wire#w5
      { S7_Templates := "SrcType := Int" } EQ_Contact(in1 := #StepDelay."Noof StepsPv", in2 := 5)
      Add(in1 := #StepDelay.StepTimeSv[1], in2 := #StepDelay.StepTimeSv[2], in3 := #StepDelay.StepTimeSv[3], in4 := #StepDelay.StepTimeSv[4], in5 := #StepDelay.StepTimePv, out => #ParaOut.Out.TimePV)
   END_RUNG
   RUNG wire#w5
      { S7_Templates := "SrcType := Int" } EQ_Contact(in1 := #StepDelay."Noof StepsPv", in2 := 6)
      Add(in1 := #StepDelay.StepTimeSv[1], in2 := #StepDelay.StepTimeSv[2], in3 := #StepDelay.StepTimeSv[3], in4 := #StepDelay.StepTimeSv[4], in5 := #StepDelay.StepTimeSv[5], in6 := #StepDelay.StepTimePv, out => #ParaOut.Out.TimePV)
   END_RUNG
   RUNG wire#w5
      { S7_Templates := "SrcType := Int" } EQ_Contact(in1 := #StepDelay."Noof StepsPv", in2 := 7)
      Add(in1 := #StepDelay.StepTimeSv[1], in2 := #StepDelay.StepTimeSv[2], in3 := #StepDelay.StepTimeSv[3], in4 := #StepDelay.StepTimeSv[4], in5 := #StepDelay.StepTimeSv[5], in6 := #StepDelay.StepTimeSv[6], in7 := #StepDelay.StepTimePv, out => #ParaOut.Out.TimePV)
   END_RUNG
   RUNG wire#w5
      { S7_Templates := "SrcType := Int" } EQ_Contact(in1 := #StepDelay."Noof StepsPv", in2 := 8)
      Add(in1 := #StepDelay.StepTimeSv[1], in2 := #StepDelay.StepTimeSv[2], in3 := #StepDelay.StepTimeSv[3], in4 := #StepDelay.StepTimeSv[4], in5 := #StepDelay.StepTimeSv[5], in6 := #StepDelay.StepTimeSv[6], in7 := #StepDelay.StepTimeSv[7], in8 := #StepDelay.StepTimePv, out => #ParaOut.Out.TimePV)
   END_RUNG
   RUNG wire#w5
      { S7_Templates := "SrcType := Int" } EQ_Contact(in1 := #StepDelay."Noof StepsPv", in2 := 9)
      Add(in1 := #StepDelay.StepTimeSv[1], in2 := #StepDelay.StepTimeSv[2], in3 := #StepDelay.StepTimeSv[3], in4 := #StepDelay.StepTimeSv[4], in5 := #StepDelay.StepTimeSv[5], in6 := #StepDelay.StepTimeSv[6], in7 := #StepDelay.StepTimeSv[7], in8 := #StepDelay.StepTimeSv[8], in9 := #StepDelay.StepTimePv, out => #ParaOut.Out.TimePV)
   END_RUNG
   RUNG wire#w5
      { S7_Templates := "SrcType := Int" } EQ_Contact(in1 := #StepDelay."Noof StepsPv", in2 := 10)
      Add(in1 := #StepDelay.StepTimeSv[1], in2 := #StepDelay.StepTimeSv[2], in3 := #StepDelay.StepTimeSv[3], in4 := #StepDelay.StepTimeSv[4], in5 := #StepDelay.StepTimeSv[5], in6 := #StepDelay.StepTimeSv[6], in7 := #StepDelay.StepTimeSv[7], in8 := #StepDelay.StepTimeSv[8], in9 := #StepDelay.StepTimeSv[9], in10 := #StepDelay.StepTimePv, out => #ParaOut.Out.TimePV)
   END_RUNG
   RUNG wire#w5
      { S7_Templates := "SrcType := Int" } EQ_Contact(in1 := #StepDelay."Noof StepsPv", in2 := 11)
      Add(in1 := #StepDelay.StepTimeSv[1], in2 := #StepDelay.StepTimeSv[2], in3 := #StepDelay.StepTimeSv[3], in4 := #StepDelay.StepTimeSv[4], in5 := #StepDelay.StepTimeSv[5], in6 := #StepDelay.StepTimeSv[6], in7 := #StepDelay.StepTimeSv[7], in8 := #StepDelay.StepTimeSv[8], in9 := #StepDelay.StepTimeSv[9], in10 := #StepDelay.StepTimeSv[10], in11 := #StepDelay.StepTimePv, out => #ParaOut.Out.TimePV)
   END_RUNG
   RUNG wire#w5
      { S7_Templates := "SrcType := Int" } EQ_Contact(in1 := #StepDelay."Noof StepsPv", in2 := 12)
      Add(in1 := #StepDelay.StepTimeSv[1], in2 := #StepDelay.StepTimeSv[2], in3 := #StepDelay.StepTimeSv[3], in4 := #StepDelay.StepTimeSv[4], in5 := #StepDelay.StepTimeSv[5], in6 := #StepDelay.StepTimeSv[6], in7 := #StepDelay.StepTimeSv[7], in8 := #StepDelay.StepTimeSv[8], in9 := #StepDelay.StepTimeSv[9], in10 := #StepDelay.StepTimeSv[10], in11 := #StepDelay.StepTimeSv[11], in12 := #StepDelay.StepTimePv, out => #ParaOut.Out.TimePV)
   END_RUNG
   RUNG wire#w5
      { S7_Templates := "SrcType := Int" } EQ_Contact(in1 := #StepDelay."Noof StepsPv", in2 := 13)
      Add(in1 := #StepDelay.StepTimeSv[1], in2 := #StepDelay.StepTimeSv[2], in3 := #StepDelay.StepTimeSv[3], in4 := #StepDelay.StepTimeSv[4], in5 := #StepDelay.StepTimeSv[5], in6 := #StepDelay.StepTimeSv[6], in7 := #StepDelay.StepTimeSv[7], in8 := #StepDelay.StepTimeSv[8], in9 := #StepDelay.StepTimeSv[9], in10 := #StepDelay.StepTimeSv[10], in11 := #StepDelay.StepTimeSv[11], in12 := #StepDelay.StepTimeSv[12], in13 := #StepDelay.StepTimePv, out => #ParaOut.Out.TimePV)
   END_RUNG
   RUNG wire#w5
      { S7_Templates := "SrcType := Int" } EQ_Contact(in1 := #StepDelay."Noof StepsPv", in2 := 14)
      Add(in1 := #StepDelay.StepTimeSv[1], in2 := #StepDelay.StepTimeSv[2], in3 := #StepDelay.StepTimeSv[3], in4 := #StepDelay.StepTimeSv[4], in5 := #StepDelay.StepTimeSv[5], in6 := #StepDelay.StepTimeSv[6], in7 := #StepDelay.StepTimeSv[7], in8 := #StepDelay.StepTimeSv[8], in9 := #StepDelay.StepTimeSv[9], in10 := #StepDelay.StepTimeSv[10], in11 := #StepDelay.StepTimeSv[11], in12 := #StepDelay.StepTimeSv[12], in13 := #StepDelay.StepTimeSv[13], in14 := #StepDelay.StepTimePv, out => #ParaOut.Out.TimePV)
   END_RUNG
   RUNG wire#w5
      { S7_Templates := "SrcType := Int" } EQ_Contact(in1 := #StepDelay."Noof StepsPv", in2 := 15)
      Add(in1 := #StepDelay.StepTimeSv[1], in2 := #StepDelay.StepTimeSv[2], in3 := #StepDelay.StepTimeSv[3], in4 := #StepDelay.StepTimeSv[4], in5 := #StepDelay.StepTimeSv[5], in6 := #StepDelay.StepTimeSv[6], in7 := #StepDelay.StepTimeSv[7], in8 := #StepDelay.StepTimeSv[8], in9 := #StepDelay.StepTimeSv[9], in10 := #StepDelay.StepTimeSv[10], in11 := #StepDelay.StepTimeSv[11], in12 := #StepDelay.StepTimeSv[12], in13 := #StepDelay.StepTimeSv[13], in14 := #StepDelay.StepTimeSv[14], in15 := #StepDelay.StepTimePv, out => #ParaOut.Out.TimePV)
   END_RUNG
   RUNG wire#w5
      { S7_Templates := "SrcType := Int" } EQ_Contact(in1 := #StepDelay."Noof StepsPv", in2 := 16)
      Add(in1 := #StepDelay.StepTimeSv[1], in2 := #StepDelay.StepTimeSv[2], in3 := #StepDelay.StepTimeSv[3], in4 := #StepDelay.StepTimeSv[4], in5 := #StepDelay.StepTimeSv[5], in6 := #StepDelay.StepTimeSv[6], in7 := #StepDelay.StepTimeSv[7], in8 := #StepDelay.StepTimeSv[8], in9 := #StepDelay.StepTimeSv[9], in10 := #StepDelay.StepTimeSv[10], in11 := #StepDelay.StepTimeSv[11], in12 := #StepDelay.StepTimeSv[12], in13 := #StepDelay.StepTimeSv[13], in14 := #StepDelay.StepTimeSv[14], in15 := #StepDelay.StepTimeSv[15], in16 := #StepDelay.StepTimePv, out => #ParaOut.Out.TimePV)
   END_RUNG
   RUNG wire#w5
      { S7_Templates := "SrcType := Int" } EQ_Contact(in1 := #StepDelay."Noof StepsPv", in2 := 17)
      Add(in1 := #StepDelay.StepTimeSv[1], in2 := #StepDelay.StepTimeSv[2], in3 := #StepDelay.StepTimeSv[3], in4 := #StepDelay.StepTimeSv[4], in5 := #StepDelay.StepTimeSv[5], in6 := #StepDelay.StepTimeSv[6], in7 := #StepDelay.StepTimeSv[7], in8 := #StepDelay.StepTimeSv[8], in9 := #StepDelay.StepTimeSv[9], in10 := #StepDelay.StepTimeSv[10], in11 := #StepDelay.StepTimeSv[11], in12 := #StepDelay.StepTimeSv[12], in13 := #StepDelay.StepTimeSv[13], in14 := #StepDelay.StepTimeSv[14], in15 := #StepDelay.StepTimeSv[15], in16 := #StepDelay.StepTimeSv[16], in17 := #StepDelay.StepTimePv, out => #ParaOut.Out.TimePV)
   END_RUNG
   RUNG wire#w2
      I_Contact( #CycleEnable )
      Move(in := 0, out1 => #ParaOut.Out.TimePV)
   END_RUNG
   RUNG wire#w1
      I_Contact( #CycleEnable )
      Move(in := 0, out1 => #ParaOut.Out.TimePV)
   END_RUNG
   // the same network as SCL:
   #_w1 := "AlwaysTRUE" AND (#StepDelay.StepTimePv >= 0);
   #_w2 := #_w1 AND (#ParaIn.PreciseEngineering.Loops <= 20);
   IF #_w2 THEN
       #ParaOut.Out.TimeSV := #StepDelay.StepTimeSv[1] + #StepDelay.StepTimeSv[2] + #StepDelay.StepTimeSv[3] + #StepDelay.StepTimeSv[4] + #StepDelay.StepTimeSv[5] + #StepDelay.StepTimeSv[6] + #StepDelay.StepTimeSv[7] + #StepDelay.StepTimeSv[8] + #StepDelay.StepTimeSv[9] + #StepDelay.StepTimeSv[10] + #StepDelay.StepTimeSv[11] + #StepDelay.StepTimeSv[12] + #StepDelay.StepTimeSv[13] + #StepDelay.StepTimeSv[14] + #StepDelay.StepTimeSv[15] + #StepDelay.StepTimeSv[16] + #StepDelay.StepTimeSv[17];
   END_IF;
   IF #_w2 AND #OverTemp THEN
       #ParaOut.Out.TimePV := #StepDelay.StepTimeSv[1] + #StepDelay.StepTimeSv[2] + #StepDelay.StepTimeSv[3] + #StepDelay.StepTimeSv[4] + #StepDelay.StepTimeSv[5] + #StepDelay.StepTimeSv[6] + #StepDelay.StepTimeSv[7] + #StepDelay.StepTimeSv[8] + #StepDelay.StepTimeSv[9] + #StepDelay.StepTimeSv[10] + #StepDelay.StepTimeSv[11] + #StepDelay.StepTimeSv[12] + #StepDelay.StepTimeSv[13] + #StepDelay.StepTimeSv[14] + #StepDelay.StepTimeSv[15] + #StepDelay.StepTimeSv[16] + #StepDelay.StepTimeSv[17];
   END_IF;
   #_w3 := #_w1 AND (#ParaIn.PreciseEngineering.Loops = 5) AND NOT #AlwaysTrue;
   IF #_w3 THEN
       #ParaOut.Out.TimeSV := #StepDelay.StepTimeSv[1] + #StepDelay.StepTimeSv[2] + #StepDelay.StepTimeSv[3] + #StepDelay.StepTimeSv[4] + #StepDelay.StepTimeSv[5];
   END_IF;
   IF #_w3 AND #OverTemp THEN
       #ParaOut.Out.TimePV := #StepDelay.StepTimeSv[1] + #StepDelay.StepTimeSv[2] + #StepDelay.StepTimeSv[3] + #StepDelay.StepTimeSv[4] + #StepDelay.StepTimeSv[5];
   END_IF;
   #_w4 := #_w1 AND #CycleEnable;
   IF #_w4 AND (#StepDelay."Noof StepsPv" = 1) THEN #ParaOut.Out.TimePV := #StepDelay.StepTimePv; END_IF;
   IF #_w4 AND (#StepDelay."Noof StepsPv" = 2) THEN
       #ParaOut.Out.TimePV := #StepDelay.StepTimeSv[1] + #StepDelay.StepTimePv;
   END_IF;
   IF #_w4 AND (#StepDelay."Noof StepsPv" = 3) THEN
       #ParaOut.Out.TimePV := #StepDelay.StepTimeSv[1] + #StepDelay.StepTimeSv[2] + #StepDelay.StepTimePv;
   END_IF;
   IF #_w4 AND (#StepDelay."Noof StepsPv" = 4) THEN
       #ParaOut.Out.TimePV := #StepDelay.StepTimeSv[1] + #StepDelay.StepTimeSv[2] + #StepDelay.StepTimeSv[3] + #StepDelay.StepTimePv;
   END_IF;
   IF #_w4 AND (#StepDelay."Noof StepsPv" = 5) THEN
       #ParaOut.Out.TimePV := #StepDelay.StepTimeSv[1] + #StepDelay.StepTimeSv[2] + #StepDelay.StepTimeSv[3] + #StepDelay.StepTimeSv[4] + #StepDelay.StepTimePv;
   END_IF;
   IF #_w4 AND (#StepDelay."Noof StepsPv" = 6) THEN
       #ParaOut.Out.TimePV := #StepDelay.StepTimeSv[1] + #StepDelay.StepTimeSv[2] + #StepDelay.StepTimeSv[3] + #StepDelay.StepTimeSv[4] + #StepDelay.StepTimeSv[5] + #StepDelay.StepTimePv;
   END_IF;
   IF #_w4 AND (#StepDelay."Noof StepsPv" = 7) THEN
       #ParaOut.Out.TimePV := #StepDelay.StepTimeSv[1] + #StepDelay.StepTimeSv[2] + #StepDelay.StepTimeSv[3] + #StepDelay.StepTimeSv[4] + #StepDelay.StepTimeSv[5] + #StepDelay.StepTimeSv[6] + #StepDelay.StepTimePv;
   END_IF;
   IF #_w4 AND (#StepDelay."Noof StepsPv" = 8) THEN
       #ParaOut.Out.TimePV := #StepDelay.StepTimeSv[1] + #StepDelay.StepTimeSv[2] + #StepDelay.StepTimeSv[3] + #StepDelay.StepTimeSv[4] + #StepDelay.StepTimeSv[5] + #StepDelay.StepTimeSv[6] + #StepDelay.StepTimeSv[7] + #StepDelay.StepTimePv;
   END_IF;
   IF #_w4 AND (#StepDelay."Noof StepsPv" = 9) THEN
       #ParaOut.Out.TimePV := #StepDelay.StepTimeSv[1] + #StepDelay.StepTimeSv[2] + #StepDelay.StepTimeSv[3] + #StepDelay.StepTimeSv[4] + #StepDelay.StepTimeSv[5] + #StepDelay.StepTimeSv[6] + #StepDelay.StepTimeSv[7] + #StepDelay.StepTimeSv[8] + #StepDelay.StepTimePv;
   END_IF;
   IF #_w4 AND (#StepDelay."Noof StepsPv" = 10) THEN
       #ParaOut.Out.TimePV := #StepDelay.StepTimeSv[1] + #StepDelay.StepTimeSv[2] + #StepDelay.StepTimeSv[3] + #StepDelay.StepTimeSv[4] + #StepDelay.StepTimeSv[5] + #StepDelay.StepTimeSv[6] + #StepDelay.StepTimeSv[7] + #StepDelay.StepTimeSv[8] + #StepDelay.StepTimeSv[9] + #StepDelay.StepTimePv;
   END_IF;
   IF #_w4 AND (#StepDelay."Noof StepsPv" = 11) THEN
       #ParaOut.Out.TimePV := #StepDelay.StepTimeSv[1] + #StepDelay.StepTimeSv[2] + #StepDelay.StepTimeSv[3] + #StepDelay.StepTimeSv[4] + #StepDelay.StepTimeSv[5] + #StepDelay.StepTimeSv[6] + #StepDelay.StepTimeSv[7] + #StepDelay.StepTimeSv[8] + #StepDelay.StepTimeSv[9] + #StepDelay.StepTimeSv[10] + #StepDelay.StepTimePv;
   END_IF;
   IF #_w4 AND (#StepDelay."Noof StepsPv" = 12) THEN
       #ParaOut.Out.TimePV := #StepDelay.StepTimeSv[1] + #StepDelay.StepTimeSv[2] + #StepDelay.StepTimeSv[3] + #StepDelay.StepTimeSv[4] + #StepDelay.StepTimeSv[5] + #StepDelay.StepTimeSv[6] + #StepDelay.StepTimeSv[7] + #StepDelay.StepTimeSv[8] + #StepDelay.StepTimeSv[9] + #StepDelay.StepTimeSv[10] + #StepDelay.StepTimeSv[11] + #StepDelay.StepTimePv;
   END_IF;
   IF #_w4 AND (#StepDelay."Noof StepsPv" = 13) THEN
       #ParaOut.Out.TimePV := #StepDelay.StepTimeSv[1] + #StepDelay.StepTimeSv[2] + #StepDelay.StepTimeSv[3] + #StepDelay.StepTimeSv[4] + #StepDelay.StepTimeSv[5] + #StepDelay.StepTimeSv[6] + #StepDelay.StepTimeSv[7] + #StepDelay.StepTimeSv[8] + #StepDelay.StepTimeSv[9] + #StepDelay.StepTimeSv[10] + #StepDelay.StepTimeSv[11] + #StepDelay.StepTimeSv[12] + #StepDelay.StepTimePv;
   END_IF;
   IF #_w4 AND (#StepDelay."Noof StepsPv" = 14) THEN
       #ParaOut.Out.TimePV := #StepDelay.StepTimeSv[1] + #StepDelay.StepTimeSv[2] + #StepDelay.StepTimeSv[3] + #StepDelay.StepTimeSv[4] + #StepDelay.StepTimeSv[5] + #StepDelay.StepTimeSv[6] + #StepDelay.StepTimeSv[7] + #StepDelay.StepTimeSv[8] + #StepDelay.StepTimeSv[9] + #StepDelay.StepTimeSv[10] + #StepDelay.StepTimeSv[11] + #StepDelay.StepTimeSv[12] + #StepDelay.StepTimeSv[13] + #StepDelay.StepTimePv;
   END_IF;
   IF #_w4 AND (#StepDelay."Noof StepsPv" = 15) THEN
       #ParaOut.Out.TimePV := #StepDelay.StepTimeSv[1] + #StepDelay.StepTimeSv[2] + #StepDelay.StepTimeSv[3] + #StepDelay.StepTimeSv[4] + #StepDelay.StepTimeSv[5] + #StepDelay.StepTimeSv[6] + #StepDelay.StepTimeSv[7] + #StepDelay.StepTimeSv[8] + #StepDelay.StepTimeSv[9] + #StepDelay.StepTimeSv[10] + #StepDelay.StepTimeSv[11] + #StepDelay.StepTimeSv[12] + #StepDelay.StepTimeSv[13] + #StepDelay.StepTimeSv[14] + #StepDelay.StepTimePv;
   END_IF;
   IF #_w4 AND (#StepDelay."Noof StepsPv" = 16) THEN
       #ParaOut.Out.TimePV := #StepDelay.StepTimeSv[1] + #StepDelay.StepTimeSv[2] + #StepDelay.StepTimeSv[3] + #StepDelay.StepTimeSv[4] + #StepDelay.StepTimeSv[5] + #StepDelay.StepTimeSv[6] + #StepDelay.StepTimeSv[7] + #StepDelay.StepTimeSv[8] + #StepDelay.StepTimeSv[9] + #StepDelay.StepTimeSv[10] + #StepDelay.StepTimeSv[11] + #StepDelay.StepTimeSv[12] + #StepDelay.StepTimeSv[13] + #StepDelay.StepTimeSv[14] + #StepDelay.StepTimeSv[15] + #StepDelay.StepTimePv;
   END_IF;
   IF #_w4 AND (#StepDelay."Noof StepsPv" = 17) THEN
       #ParaOut.Out.TimePV := #StepDelay.StepTimeSv[1] + #StepDelay.StepTimeSv[2] + #StepDelay.StepTimeSv[3] + #StepDelay.StepTimeSv[4] + #StepDelay.StepTimeSv[5] + #StepDelay.StepTimeSv[6] + #StepDelay.StepTimeSv[7] + #StepDelay.StepTimeSv[8] + #StepDelay.StepTimeSv[9] + #StepDelay.StepTimeSv[10] + #StepDelay.StepTimeSv[11] + #StepDelay.StepTimeSv[12] + #StepDelay.StepTimeSv[13] + #StepDelay.StepTimeSv[14] + #StepDelay.StepTimeSv[15] + #StepDelay.StepTimeSv[16] + #StepDelay.StepTimePv;
   END_IF;
   IF #_w1 AND NOT #CycleEnable THEN #ParaOut.Out.TimePV := 0; END_IF;
   IF "AlwaysTRUE" AND NOT #CycleEnable THEN #ParaOut.Out.TimePV := 0; END_IF;
END_REGION

REGION Network 12: #StepDelay
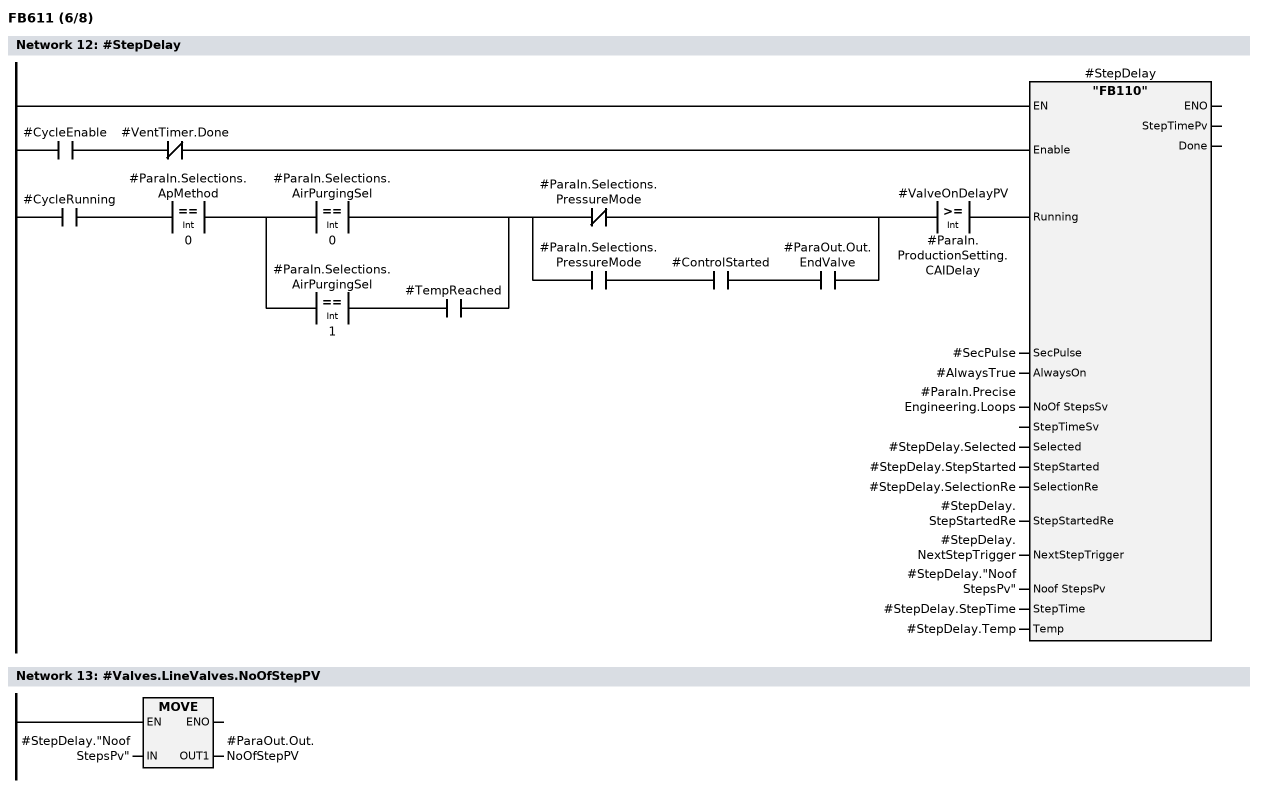
   RUNG wire#powerrail
      #StepDelay(Enable := wire#w1, Running := wire#w5, SecPulse := #SecPulse, AlwaysOn := #AlwaysTrue, "NoOf StepsSv" := #ParaIn.PreciseEngineering.Loops, StepTimeSv :=, Selected := #StepDelay.Selected, StepStarted := #StepDelay.StepStarted, SelectionRe := #StepDelay.SelectionRe, StepStartedRe := #StepDelay.StepStartedRe, NextStepTrigger := #StepDelay.NextStepTrigger, "Noof StepsPv" := #StepDelay."Noof StepsPv", StepTime := #StepDelay.StepTime, Temp := #StepDelay.Temp, StepTimePv =>, Done =>)
   END_RUNG
   RUNG wire#powerrail
      Contact( #CycleEnable )
      I_Contact( #VentTimer.Done )
   END_RUNG wire#w1
   RUNG wire#powerrail
      Contact( #CycleRunning )
      { S7_Templates := "SrcType := Int" } EQ_Contact(in1 := #ParaIn.Selections.ApMethod, in2 := 0)
      wire#w2
      { S7_Templates := "SrcType := Int" } EQ_Contact(in1 := #ParaIn.Selections.AirPurgingSel, in2 := 0)
      wire#w3
      I_Contact( #ParaIn.Selections.PressureMode )
      wire#w4
      { S7_Templates := "SrcType := Int" } GE_Contact(in1 := #ValveOnDelayPV, in2 := #ParaIn.ProductionSetting.CAIDelay)
   END_RUNG wire#w5
   RUNG wire#w2
      { S7_Templates := "SrcType := Int" } EQ_Contact(in1 := #ParaIn.Selections.AirPurgingSel, in2 := 1)
      Contact( #TempReached )
   END_RUNG wire#w3
   RUNG wire#w3
      Contact( #ParaIn.Selections.PressureMode )
      Contact( #ControlStarted )
      Contact( #ParaOut.Out.EndValve )
   END_RUNG wire#w4
   // the same network as SCL:
   #StepDelay(Enable := #CycleEnable AND NOT #VentTimer.Done,   // "FB110"
              Running := #CycleRunning AND (#ParaIn.Selections.ApMethod = 0) AND ((#ParaIn.Selections.AirPurgingSel = 0) OR ((#ParaIn.Selections.AirPurgingSel = 1) AND #TempReached)) AND (NOT #ParaIn.Selections.PressureMode OR (#ParaIn.Selections.PressureMode AND #ControlStarted AND #ParaOut.Out.EndValve)) AND (#ValveOnDelayPV >= #ParaIn.ProductionSetting.CAIDelay),
              SecPulse := #SecPulse,
              AlwaysOn := #AlwaysTrue,
              "NoOf StepsSv" := #ParaIn.PreciseEngineering.Loops,
              Selected := #StepDelay.Selected,
              StepStarted := #StepDelay.StepStarted,
              SelectionRe := #StepDelay.SelectionRe,
              StepStartedRe := #StepDelay.StepStartedRe,
              NextStepTrigger := #StepDelay.NextStepTrigger,
              "Noof StepsPv" := #StepDelay."Noof StepsPv",
              StepTime := #StepDelay.StepTime,
              Temp := #StepDelay.Temp);
END_REGION

REGION Network 13: #Valves.LineValves.NoOfStepPV
   RUNG wire#powerrail
      Move(in := #StepDelay."Noof StepsPv", out1 => #ParaOut.Out.NoOfStepPV)
   END_RUNG
   // the same network as SCL:
   #ParaOut.Out.NoOfStepPV := #StepDelay."Noof StepsPv";
END_REGION

REGION Network 14: Loop Outputs
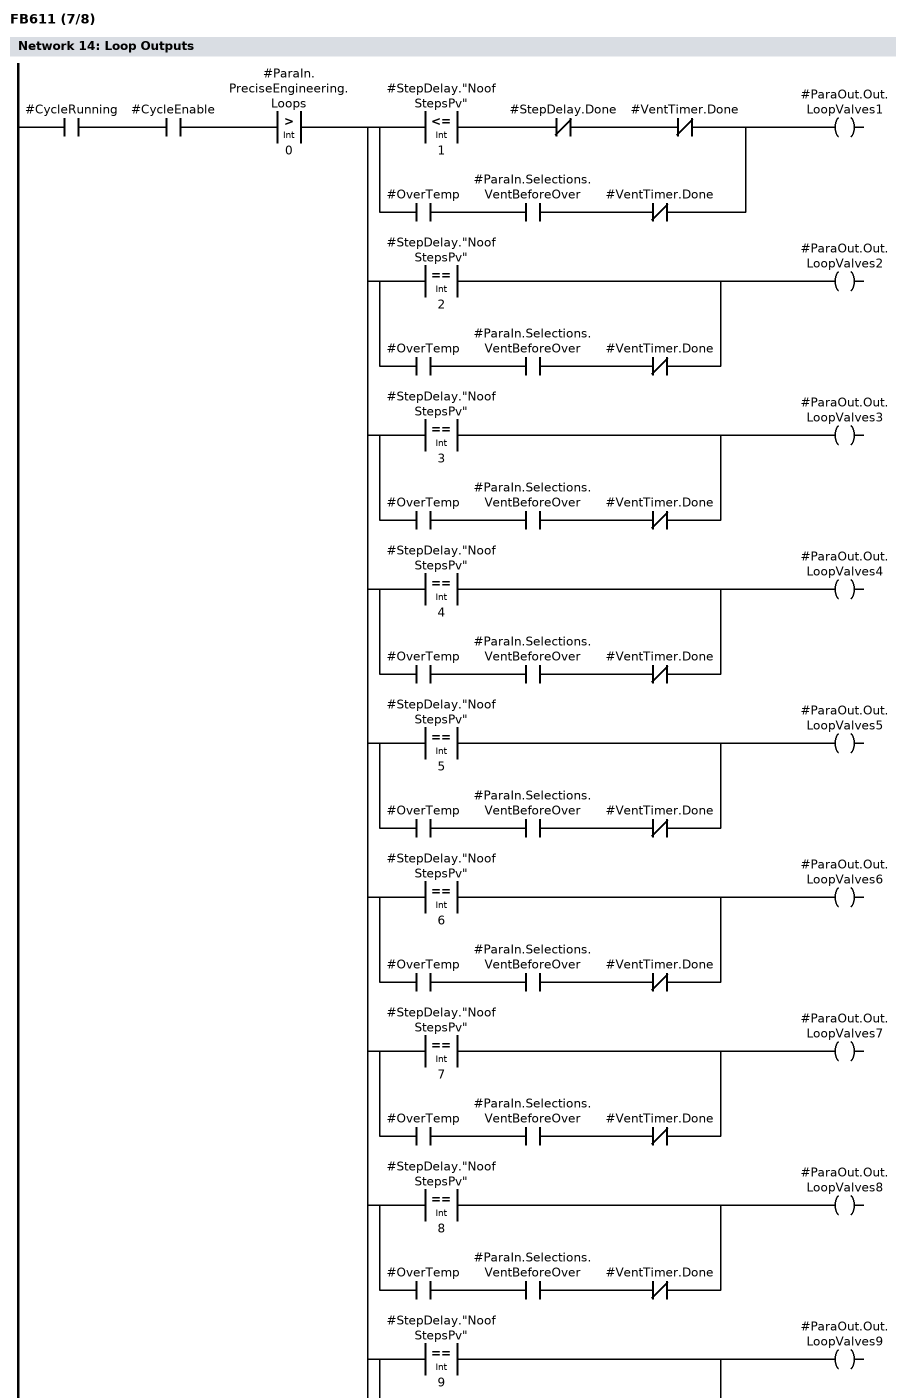
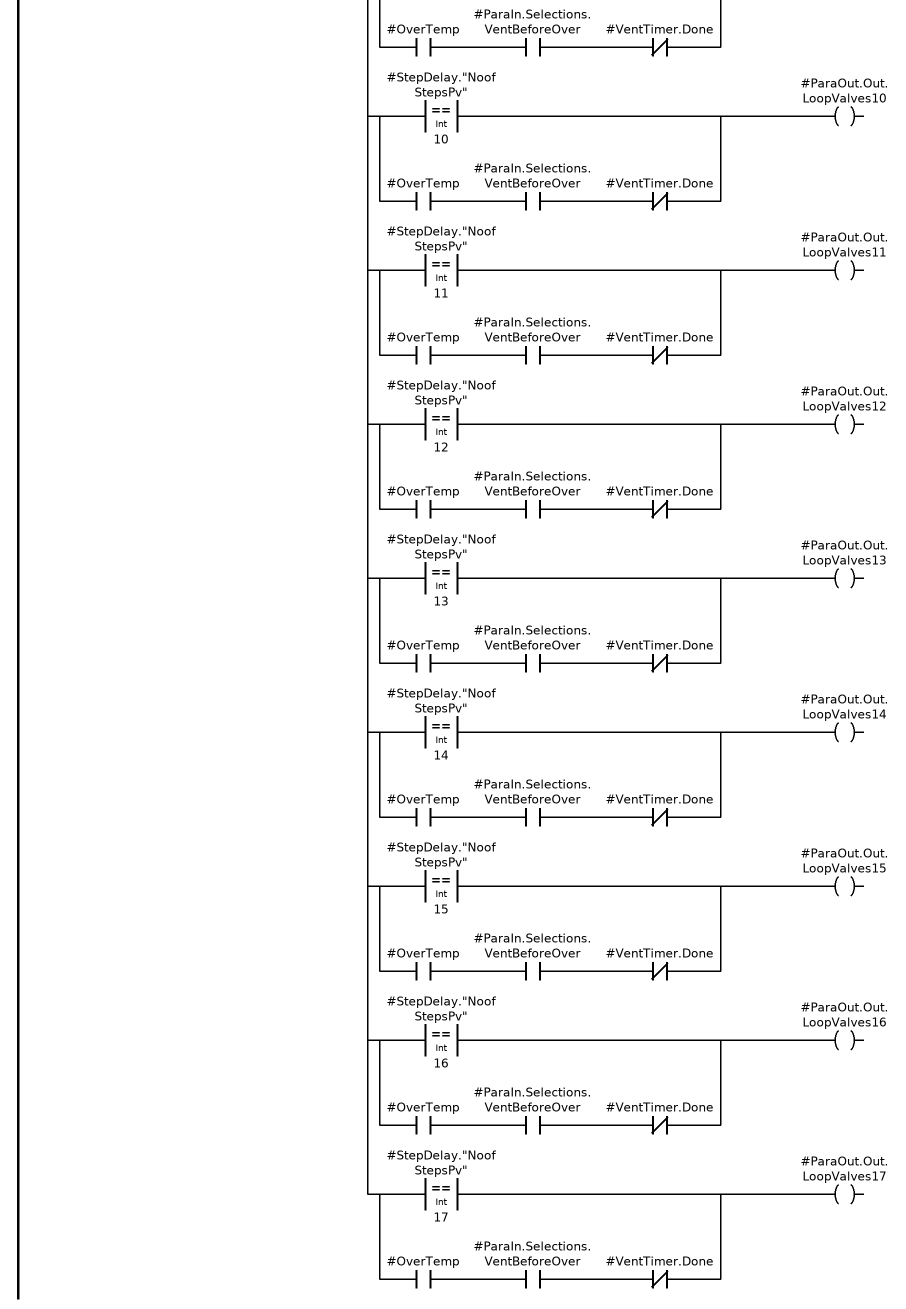
   RUNG wire#powerrail
      Contact( #CycleRunning )
      Contact( #CycleEnable )
      { S7_Templates := "SrcType := Int" } GT_Contact(in1 := #ParaIn.PreciseEngineering.Loops, in2 := 0)
      wire#w1
      { S7_Templates := "SrcType := Int" } LE_Contact(in1 := #StepDelay."Noof StepsPv", in2 := 1)
      I_Contact( #StepDelay.Done )
      I_Contact( #VentTimer.Done )
      wire#w2
      Coil( #ParaOut.Out.LoopValves1 )
   END_RUNG
   RUNG wire#w1
      Contact( #OverTemp )
      Contact( #ParaIn.Selections.VentBeforeOver )
      I_Contact( #VentTimer.Done )
   END_RUNG wire#w2
   RUNG wire#w1
      { S7_Templates := "SrcType := Int" } EQ_Contact(in1 := #StepDelay."Noof StepsPv", in2 := 2)
      wire#w3
      Coil( #ParaOut.Out.LoopValves2 )
   END_RUNG
   RUNG wire#w1
      Contact( #OverTemp )
      Contact( #ParaIn.Selections.VentBeforeOver )
      I_Contact( #VentTimer.Done )
   END_RUNG wire#w3
   RUNG wire#w1
      { S7_Templates := "SrcType := Int" } EQ_Contact(in1 := #StepDelay."Noof StepsPv", in2 := 3)
      wire#w4
      Coil( #ParaOut.Out.LoopValves3 )
   END_RUNG
   RUNG wire#w1
      Contact( #OverTemp )
      Contact( #ParaIn.Selections.VentBeforeOver )
      I_Contact( #VentTimer.Done )
   END_RUNG wire#w4
   RUNG wire#w1
      { S7_Templates := "SrcType := Int" } EQ_Contact(in1 := #StepDelay."Noof StepsPv", in2 := 4)
      wire#w5
      Coil( #ParaOut.Out.LoopValves4 )
   END_RUNG
   RUNG wire#w1
      Contact( #OverTemp )
      Contact( #ParaIn.Selections.VentBeforeOver )
      I_Contact( #VentTimer.Done )
   END_RUNG wire#w5
   RUNG wire#w1
      { S7_Templates := "SrcType := Int" } EQ_Contact(in1 := #StepDelay."Noof StepsPv", in2 := 5)
      wire#w6
      Coil( #ParaOut.Out.LoopValves5 )
   END_RUNG
   RUNG wire#w1
      Contact( #OverTemp )
      Contact( #ParaIn.Selections.VentBeforeOver )
      I_Contact( #VentTimer.Done )
   END_RUNG wire#w6
   RUNG wire#w1
      { S7_Templates := "SrcType := Int" } EQ_Contact(in1 := #StepDelay."Noof StepsPv", in2 := 6)
      wire#w7
      Coil( #ParaOut.Out.LoopValves6 )
   END_RUNG
   RUNG wire#w1
      Contact( #OverTemp )
      Contact( #ParaIn.Selections.VentBeforeOver )
      I_Contact( #VentTimer.Done )
   END_RUNG wire#w7
   RUNG wire#w1
      { S7_Templates := "SrcType := Int" } EQ_Contact(in1 := #StepDelay."Noof StepsPv", in2 := 7)
      wire#w8
      Coil( #ParaOut.Out.LoopValves7 )
   END_RUNG
   RUNG wire#w1
      Contact( #OverTemp )
      Contact( #ParaIn.Selections.VentBeforeOver )
      I_Contact( #VentTimer.Done )
   END_RUNG wire#w8
   RUNG wire#w1
      { S7_Templates := "SrcType := Int" } EQ_Contact(in1 := #StepDelay."Noof StepsPv", in2 := 8)
      wire#w9
      Coil( #ParaOut.Out.LoopValves8 )
   END_RUNG
   RUNG wire#w1
      Contact( #OverTemp )
      Contact( #ParaIn.Selections.VentBeforeOver )
      I_Contact( #VentTimer.Done )
   END_RUNG wire#w9
   RUNG wire#w1
      { S7_Templates := "SrcType := Int" } EQ_Contact(in1 := #StepDelay."Noof StepsPv", in2 := 9)
      wire#w10
      Coil( #ParaOut.Out.LoopValves9 )
   END_RUNG
   RUNG wire#w1
      Contact( #OverTemp )
      Contact( #ParaIn.Selections.VentBeforeOver )
      I_Contact( #VentTimer.Done )
   END_RUNG wire#w10
   RUNG wire#w1
      { S7_Templates := "SrcType := Int" } EQ_Contact(in1 := #StepDelay."Noof StepsPv", in2 := 10)
      wire#w11
      Coil( #ParaOut.Out.LoopValves10 )
   END_RUNG
   RUNG wire#w1
      Contact( #OverTemp )
      Contact( #ParaIn.Selections.VentBeforeOver )
      I_Contact( #VentTimer.Done )
   END_RUNG wire#w11
   RUNG wire#w1
      { S7_Templates := "SrcType := Int" } EQ_Contact(in1 := #StepDelay."Noof StepsPv", in2 := 11)
      wire#w12
      Coil( #ParaOut.Out.LoopValves11 )
   END_RUNG
   RUNG wire#w1
      Contact( #OverTemp )
      Contact( #ParaIn.Selections.VentBeforeOver )
      I_Contact( #VentTimer.Done )
   END_RUNG wire#w12
   RUNG wire#w1
      { S7_Templates := "SrcType := Int" } EQ_Contact(in1 := #StepDelay."Noof StepsPv", in2 := 12)
      wire#w13
      Coil( #ParaOut.Out.LoopValves12 )
   END_RUNG
   RUNG wire#w1
      Contact( #OverTemp )
      Contact( #ParaIn.Selections.VentBeforeOver )
      I_Contact( #VentTimer.Done )
   END_RUNG wire#w13
   RUNG wire#w1
      { S7_Templates := "SrcType := Int" } EQ_Contact(in1 := #StepDelay."Noof StepsPv", in2 := 13)
      wire#w14
      Coil( #ParaOut.Out.LoopValves13 )
   END_RUNG
   RUNG wire#w1
      Contact( #OverTemp )
      Contact( #ParaIn.Selections.VentBeforeOver )
      I_Contact( #VentTimer.Done )
   END_RUNG wire#w14
   RUNG wire#w1
      { S7_Templates := "SrcType := Int" } EQ_Contact(in1 := #StepDelay."Noof StepsPv", in2 := 14)
      wire#w15
      Coil( #ParaOut.Out.LoopValves14 )
   END_RUNG
   RUNG wire#w1
      Contact( #OverTemp )
      Contact( #ParaIn.Selections.VentBeforeOver )
      I_Contact( #VentTimer.Done )
   END_RUNG wire#w15
   RUNG wire#w1
      { S7_Templates := "SrcType := Int" } EQ_Contact(in1 := #StepDelay."Noof StepsPv", in2 := 15)
      wire#w16
      Coil( #ParaOut.Out.LoopValves15 )
   END_RUNG
   RUNG wire#w1
      Contact( #OverTemp )
      Contact( #ParaIn.Selections.VentBeforeOver )
      I_Contact( #VentTimer.Done )
   END_RUNG wire#w16
   RUNG wire#w1
      { S7_Templates := "SrcType := Int" } EQ_Contact(in1 := #StepDelay."Noof StepsPv", in2 := 16)
      wire#w17
      Coil( #ParaOut.Out.LoopValves16 )
   END_RUNG
   RUNG wire#w1
      Contact( #OverTemp )
      Contact( #ParaIn.Selections.VentBeforeOver )
      I_Contact( #VentTimer.Done )
   END_RUNG wire#w17
   RUNG wire#w1
      { S7_Templates := "SrcType := Int" } EQ_Contact(in1 := #StepDelay."Noof StepsPv", in2 := 17)
      wire#w18
      Coil( #ParaOut.Out.LoopValves17 )
   END_RUNG
   RUNG wire#w1
      Contact( #OverTemp )
      Contact( #ParaIn.Selections.VentBeforeOver )
      I_Contact( #VentTimer.Done )
   END_RUNG wire#w18
   // the same network as SCL:
   #_w1 := #CycleRunning AND #CycleEnable AND (#ParaIn.PreciseEngineering.Loops > 0);
   #ParaOut.Out.LoopValves1 := #_w1 AND (((#StepDelay."Noof StepsPv" <= 1) AND NOT #StepDelay.Done AND NOT #VentTimer.Done) OR (#OverTemp AND #ParaIn.Selections.VentBeforeOver AND NOT #VentTimer.Done));
   #ParaOut.Out.LoopValves2 := #_w1 AND ((#StepDelay."Noof StepsPv" = 2) OR (#OverTemp AND #ParaIn.Selections.VentBeforeOver AND NOT #VentTimer.Done));
   #ParaOut.Out.LoopValves3 := #_w1 AND ((#StepDelay."Noof StepsPv" = 3) OR (#OverTemp AND #ParaIn.Selections.VentBeforeOver AND NOT #VentTimer.Done));
   #ParaOut.Out.LoopValves4 := #_w1 AND ((#StepDelay."Noof StepsPv" = 4) OR (#OverTemp AND #ParaIn.Selections.VentBeforeOver AND NOT #VentTimer.Done));
   #ParaOut.Out.LoopValves5 := #_w1 AND ((#StepDelay."Noof StepsPv" = 5) OR (#OverTemp AND #ParaIn.Selections.VentBeforeOver AND NOT #VentTimer.Done));
   #ParaOut.Out.LoopValves6 := #_w1 AND ((#StepDelay."Noof StepsPv" = 6) OR (#OverTemp AND #ParaIn.Selections.VentBeforeOver AND NOT #VentTimer.Done));
   #ParaOut.Out.LoopValves7 := #_w1 AND ((#StepDelay."Noof StepsPv" = 7) OR (#OverTemp AND #ParaIn.Selections.VentBeforeOver AND NOT #VentTimer.Done));
   #ParaOut.Out.LoopValves8 := #_w1 AND ((#StepDelay."Noof StepsPv" = 8) OR (#OverTemp AND #ParaIn.Selections.VentBeforeOver AND NOT #VentTimer.Done));
   #ParaOut.Out.LoopValves9 := #_w1 AND ((#StepDelay."Noof StepsPv" = 9) OR (#OverTemp AND #ParaIn.Selections.VentBeforeOver AND NOT #VentTimer.Done));
   #ParaOut.Out.LoopValves10 := #_w1 AND ((#StepDelay."Noof StepsPv" = 10) OR (#OverTemp AND #ParaIn.Selections.VentBeforeOver AND NOT #VentTimer.Done));
   #ParaOut.Out.LoopValves11 := #_w1 AND ((#StepDelay."Noof StepsPv" = 11) OR (#OverTemp AND #ParaIn.Selections.VentBeforeOver AND NOT #VentTimer.Done));
   #ParaOut.Out.LoopValves12 := #_w1 AND ((#StepDelay."Noof StepsPv" = 12) OR (#OverTemp AND #ParaIn.Selections.VentBeforeOver AND NOT #VentTimer.Done));
   #ParaOut.Out.LoopValves13 := #_w1 AND ((#StepDelay."Noof StepsPv" = 13) OR (#OverTemp AND #ParaIn.Selections.VentBeforeOver AND NOT #VentTimer.Done));
   #ParaOut.Out.LoopValves14 := #_w1 AND ((#StepDelay."Noof StepsPv" = 14) OR (#OverTemp AND #ParaIn.Selections.VentBeforeOver AND NOT #VentTimer.Done));
   #ParaOut.Out.LoopValves15 := #_w1 AND ((#StepDelay."Noof StepsPv" = 15) OR (#OverTemp AND #ParaIn.Selections.VentBeforeOver AND NOT #VentTimer.Done));
   #ParaOut.Out.LoopValves16 := #_w1 AND ((#StepDelay."Noof StepsPv" = 16) OR (#OverTemp AND #ParaIn.Selections.VentBeforeOver AND NOT #VentTimer.Done));
   #ParaOut.Out.LoopValves17 := #_w1 AND ((#StepDelay."Noof StepsPv" = 17) OR (#OverTemp AND #ParaIn.Selections.VentBeforeOver AND NOT #VentTimer.Done));
END_REGION

REGION Network 15: Reset
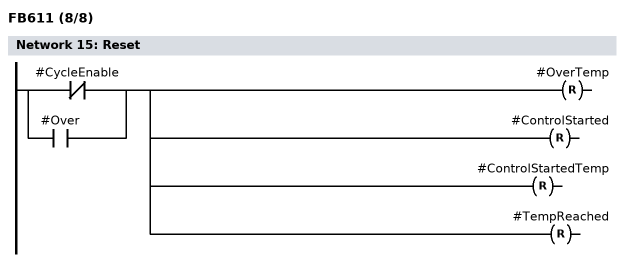
   RUNG wire#powerrail
      I_Contact( #CycleEnable )
      wire#w1
      R_Coil( #OverTemp )
   END_RUNG
   RUNG wire#powerrail
      Contact( #Over )
   END_RUNG wire#w1
   RUNG wire#w1
      R_Coil( #ControlStarted )
   END_RUNG
   RUNG wire#w1
      R_Coil( #ControlStartedTemp )
   END_RUNG
   RUNG wire#w1
      R_Coil( #TempReached )
   END_RUNG
   // the same network as SCL:
   IF NOT #CycleEnable OR #Over THEN
       #OverTemp := FALSE;
       #ControlStarted := FALSE;
       #ControlStartedTemp := FALSE;
       #TempReached := FALSE;
   END_IF;
END_REGION
END_FUNCTION_BLOCK
